LIN {X 0,Y 523.493,Z 544.016,A -85,B 0,C 180,E1 -4763.834,E2 -4763.834} C_VEL
LIN {X 0,Y 523.412,Z 548.835,A -85,B 0,C 180,E1 -4764.993,E2 -4764.993} C_VEL
LIN {X 0,Y 523.475,Z 552.534,A -85,B 0,C 180,E1 -4766.151,E2 -4766.151} C_VEL
LIN {X 0,Y 523.423,Z 554.433,A -85,B 0,C 180,E1 -4766.921,E2 -4766.921} C_VEL
LIN {X 0,Y 523.357,Z 555.854,A -85,B 0,C 180,E1 -4767.691,E2 -4767.691} C_VEL
LIN {X 0,Y 523.305,Z 557.491,A -85,B 0,C 180,E1 -4769.23,E2 -4769.23} C_VEL
LIN {X 0,Y 523.307,Z 557.714,A -85,B 0,C 180,E1 -4770,E2 -4770} C_VEL
LIN {X 0,Y 523.305,Z 557.495,A -85,B 0,C 180,E1 -4770.769,E2 -4770.769} C_VEL
LIN {X 0,Y 523.356,Z 555.866,A -85,B 0,C 180,E1 -4772.308,E2 -4772.308} C_VEL
LIN {X 0,Y 523.423,Z 554.448,A -85,B 0,C 180,E1 -4773.078,E2 -4773.078} C_VEL
LIN {X 0,Y 523.442,Z 551.453,A -85,B 0,C 180,E1 -4774.234,E2 -4774.234} C_VEL
LIN {X 0,Y 523.464,Z 547.399,A -85,B 0,C 180,E1 -4775.392,E2 -4775.392} C_VEL
LIN {X 0,Y 523.516,Z 542.074,A -85,B 0,C 180,E1 -4776.574,E2 -4776.574} C_VEL
LIN {X 0,Y 523.617,Z 535.63,A -85,B 0,C 180,E1 -4777.713,E2 -4777.713} C_VEL
LIN {X 0,Y 523.804,Z 527.471,A -85,B 0,C 180,E1 -4778.876,E2 -4778.876} C_VEL
LIN {X 0,Y 523.991,Z 519.167,A -85,B 0,C 180,E1 -4779.846,E2 -4779.846} C_VEL
LIN {X 0,Y 524.24,Z 509.058,A -85,B 0,C 180,E1 -4780.817,E2 -4780.817} C_VEL
LIN {X 0,Y 524.542,Z 497.688,A -85,B 0,C 180,E1 -4781.69,E2 -4781.69} C_VEL
LIN {X 0,Y 524.792,Z 486.52,A -85,B 0,C 180,E1 -4782.372,E2 -4782.372} C_VEL
LIN {X 0,Y 525.029,Z 475.334,A -85,B 0,C 180,E1 -4782.907,E2 -4782.907} C_VEL
LIN {X 0,Y 525.268,Z 462.202,A -85,B 0,C 180,E1 -4783.368,E2 -4783.368} C_VEL
LIN {X 0,Y 525.476,Z 449.138,A -85,B 0,C 180,E1 -4783.658,E2 -4783.658} C_VEL
LIN {X 0,Y 525.785,Z 353.498,A -85,B 0,C 180,E1 -4784.975,E2 -4784.975} C_VEL
LIN {X 0,Y 524.395,Z 341.8,A -85,B 0,C 180,E1 -4785.201,E2 -4785.201} C_VEL
LIN {X 0,Y 524.831,Z 315.783,A -85,B 0,C 180,E1 -4788.301,E2 -4788.301} C_VEL
LIN {X 0,Y 525.302,Z 288.649,A -85,B 0,C 180,E1 -4791.587,E2 -4791.587} C_VEL
LIN {X 0,Y 525.7,Z 266.745,A -85,B 0,C 180,E1 -4794.272,E2 -4794.272} C_VEL
LIN {X 0,Y 525.943,Z 250.474,A -85,B 0,C 180,E1 -4796.291,E2 -4796.291} C_VEL
LIN {X 0,Y 523.9,Z 240.345,A -85,B 0,C 180,E1 -4797.674,E2 -4797.674} C_VEL
LIN {X 0,Y 523.893,Z 240.226,A -85,B 0,C 180,E1 -4800.845,E2 -4800.845} C_VEL
LIN {X 0,Y 523.92,Z 240.225,A -85,B 0,C 180,E1 -4803.728,E2 -4803.728} C_VEL
LIN {X 0,Y 523.851,Z 240.227,A -85,B 0,C 180,E1 -4806.393,E2 -4806.393} C_VEL
LIN {X 0,Y 523.883,Z 240.228,A -85,B 0,C 180,E1 -4809.087,E2 -4809.087} C_VEL
LIN {X 0,Y 523.879,Z 240.223,A -85,B 0,C 180,E1 -4812.125,E2 -4812.125} C_VEL
LIN {X 0,Y 523.922,Z 240.226,A -85,B 0,C 180,E1 -4815.311,E2 -4815.311} C_VEL
LIN {X 0,Y 523.904,Z 240.222,A -85,B 0,C 180,E1 -4818.694,E2 -4818.694} C_VEL
LIN {X 0,Y 523.889,Z 240.222,A -85,B 0,C 180,E1 -4821.896,E2 -4821.896} C_VEL
LIN {X 0,Y 523.902,Z 240.227,A -85,B 0,C 180,E1 -4824.912,E2 -4824.912} C_VEL
LIN {X 0,Y 523.887,Z 240.223,A -85,B 0,C 180,E1 -4827.686,E2 -4827.686} C_VEL
LIN {X 0,Y 523.918,Z 240.223,A -85,B 0,C 180,E1 -4830.681,E2 -4830.681} C_VEL
LIN {X 0,Y 523.87,Z 240.225,A -85,B 0,C 180,E1 -4833.723,E2 -4833.723} C_VEL
LIN {X 0,Y 523.893,Z 240.223,A -85,B 0,C 180,E1 -4836.269,E2 -4836.269} C_VEL
LIN {X 0,Y 523.916,Z 240.226,A -85,B 0,C 180,E1 -4838.765,E2 -4838.765} C_VEL
LIN {X 0,Y 523.913,Z 240.222,A -85,B 0,C 180,E1 -4841.219,E2 -4841.219} C_VEL
LIN {X 0,Y 523.874,Z 240.224,A -85,B 0,C 180,E1 -4843.637,E2 -4843.637} C_VEL
LIN {X 0,Y 523.894,Z 240.222,A -85,B 0,C 180,E1 -4846.027,E2 -4846.027} C_VEL
LIN {X 0,Y 523.999,Z 240.213,A -85,B 0,C 180,E1 -4848.394,E2 -4848.394} C_VEL
LIN {X 0,Y 523.941,Z 240.215,A -85,B 0,C 180,E1 -4851.515,E2 -4851.515} C_VEL
LIN {X 0,Y 524.014,Z 240.216,A -85,B 0,C 180,E1 -4854.613,E2 -4854.613} C_VEL
LIN {X 0,Y 524.083,Z 240.198,A -85,B 0,C 180,E1 -4857.695,E2 -4857.695} C_VEL
LIN {X 0,Y 524.104,Z 240.2,A -85,B 0,C 180,E1 -4860.769,E2 -4860.769} C_VEL
LIN {X 0,Y 523.984,Z 240.211,A -85,B 0,C 180,E1 -4863.076,E2 -4863.076} C_VEL
LIN {X 0,Y 523.987,Z 240.215,A -85,B 0,C 180,E1 -4866.16,E2 -4866.16} C_VEL
LIN {X 0,Y 523.927,Z 240.217,A -85,B 0,C 180,E1 -4869.263,E2 -4869.263} C_VEL
LIN {X 0,Y 523.933,Z 240.224,A -85,B 0,C 180,E1 -4872.394,E2 -4872.394} C_VEL
LIN {X 0,Y 523.908,Z 240.22,A -85,B 0,C 180,E1 -4875.563,E2 -4875.563} C_VEL
LIN {X 0,Y 523.901,Z 240.226,A -85,B 0,C 180,E1 -4877.972,E2 -4877.972} C_VEL
LIN {X 0,Y 523.937,Z 240.221,A -85,B 0,C 180,E1 -4880.412,E2 -4880.412} C_VEL
LIN {X 0,Y 523.895,Z 240.222,A -85,B 0,C 180,E1 -4882.895,E2 -4882.895} C_VEL
LIN {X 0,Y 523.884,Z 240.224,A -85,B 0,C 180,E1 -4885.423,E2 -4885.423} C_VEL
LIN {X 0,Y 523.884,Z 240.231,A -85,B 0,C 180,E1 -4888.004,E2 -4888.004} C_VEL
LIN {X 0,Y 523.897,Z 240.221,A -85,B 0,C 180,E1 -4890.849,E2 -4890.849} C_VEL
LIN {X 0,Y 523.916,Z 240.224,A -85,B 0,C 180,E1 -4893.73,E2 -4893.73} C_VEL
LIN {X 0,Y 523.85,Z 240.229,A -85,B 0,C 180,E1 -4896.396,E2 -4896.396} C_VEL
LIN {X 0,Y 523.884,Z 240.223,A -85,B 0,C 180,E1 -4899.089,E2 -4899.089} C_VEL
LIN {X 0,Y 523.878,Z 240.228,A -85,B 0,C 180,E1 -4902.127,E2 -4902.127} C_VEL
LIN {X 0,Y 523.925,Z 240.22,A -85,B 0,C 180,E1 -4905.313,E2 -4905.313} C_VEL
LIN {X 0,Y 523.869,Z 240.225,A -85,B 0,C 180,E1 -4906.913,E2 -4906.913} C_VEL
LIN {X 0,Y 523.186,Z 240.316,A -85,B 0,C 180,E1 -4907.555,E2 -4907.555} C_VEL
LIN {X 0,Y 520.325,Z 240.672,A -85,B 0,C 180,E1 -4908.596,E2 -4908.596} C_VEL
LIN {X 0,Y 517.925,Z 240.97,A -85,B 0,C 180,E1 -4909.435,E2 -4909.435} C_VEL
LIN {X 0,Y 516.905,Z 241.096,A -85,B 0,C 180,E1 -4910.083,E2 -4910.083} C_VEL
LIN {X 0,Y 516.828,Z 241.103,A -85,B 0,C 180,E1 -4910.302,E2 -4910.302} C_VEL
LIN {X 0,Y 516.826,Z 241.103,A -85,B 0,C 180,E1 -4912.272,E2 -4912.272} C_VEL
LIN {X 0,Y 516.848,Z 241.102,A -85,B 0,C 180,E1 -4915.174,E2 -4915.174} C_VEL
LIN {X 0,Y 516.843,Z 241.103,A -85,B 0,C 180,E1 -4917.974,E2 -4917.974} C_VEL
LIN {X 0,Y 516.833,Z 241.101,A -85,B 0,C 180,E1 -4920.691,E2 -4920.691} C_VEL
LIN {X 0,Y 516.825,Z 241.109,A -85,B 0,C 180,E1 -4923.338,E2 -4923.338} C_VEL
LIN {X 0,Y 516.868,Z 241.099,A -85,B 0,C 180,E1 -4925.927,E2 -4925.927} C_VEL
LIN {X 0,Y 516.864,Z 241.097,A -85,B 0,C 180,E1 -4928.462,E2 -4928.462} C_VEL
LIN {X 0,Y 516.867,Z 241.1,A -85,B 0,C 180,E1 -4930.954,E2 -4930.954} C_VEL
LIN {X 0,Y 516.871,Z 241.104,A -85,B 0,C 180,E1 -4933.41,E2 -4933.41} C_VEL
LIN {X 0,Y 516.851,Z 241.1,A -85,B 0,C 180,E1 -4935.833,E2 -4935.833} C_VEL
LIN {X 0,Y 516.927,Z 241.09,A -85,B 0,C 180,E1 -4938.233,E2 -4938.233} C_VEL
LIN {X 0,Y 516.912,Z 241.1,A -85,B 0,C 180,E1 -4941.399,E2 -4941.399} C_VEL
LIN {X 0,Y 516.947,Z 241.206,A -85,B 0,C 180,E1 -4942.796,E2 -4942.796} C_VEL
LIN {X 0,Y 517.133,Z 242.04,A -85,B 0,C 180,E1 -4942.932,E2 -4942.932} C_VEL
LIN {X 0,Y 519.13,Z 247.934,A -85,B 0,C 180,E1 -4943.099,E2 -4943.099} C_VEL
LIN {X 0,Y 518.754,Z 330.215,A -85,B 0,C 180,E1 -4944.266,E2 -4944.266} C_VEL
LIN {X 0,Y 518.651,Z 343.83,A -85,B 0,C 180,E1 -4944.631,E2 -4944.631} C_VEL
LIN {X 0,Y 518.471,Z 356.587,A -85,B 0,C 180,E1 -4945.141,E2 -4945.141} C_VEL
LIN {X 0,Y 518.216,Z 368.942,A -85,B 0,C 180,E1 -4945.82,E2 -4945.82} C_VEL
LIN {X 0,Y 517.934,Z 379.943,A -85,B 0,C 180,E1 -4946.597,E2 -4946.597} C_VEL
LIN {X 0,Y 517.629,Z 389.885,A -85,B 0,C 180,E1 -4947.471,E2 -4947.471} C_VEL
LIN {X 0,Y 517.387,Z 398.828,A -85,B 0,C 180,E1 -4948.444,E2 -4948.444} C_VEL
LIN {X 0,Y 517.114,Z 407.548,A -85,B 0,C 180,E1 -4949.611,E2 -4949.611} C_VEL
LIN {X 0,Y 516.887,Z 414.584,A -85,B 0,C 180,E1 -4950.779,E2 -4950.779} C_VEL
LIN {X 0,Y 516.65,Z 420.23,A -85,B 0,C 180,E1 -4951.949,E2 -4951.949} C_VEL
LIN {X 0,Y 516.586,Z 424.66,A -85,B 0,C 180,E1 -4953.12,E2 -4953.12} C_VEL
LIN {X 0,Y 516.538,Z 427.004,A -85,B 0,C 180,E1 -4953.901,E2 -4953.901} C_VEL
LIN {X 0,Y 516.551,Z 428.921,A -85,B 0,C 180,E1 -4954.683,E2 -4954.683} C_VEL
LIN {X 0,Y 516.512,Z 430.446,A -85,B 0,C 180,E1 -4955.466,E2 -4955.466} C_VEL
LIN {X 0,Y 516.491,Z 431.912,A -85,B 0,C 180,E1 -4956.619,E2 -4956.619} C_VEL
LIN {X 0,Y 516.447,Z 432.547,A -85,B 0,C 180,E1 -4957.821,E2 -4957.821} C_VEL
LIN {X 0,Y 516.429,Z 432.486,A -85,B 0,C 180,E1 -4958.61,E2 -4958.61} C_VEL
LIN {X 0,Y 516.434,Z 432.004,A -85,B 0,C 180,E1 -4959.399,E2 -4959.399} C_VEL
LIN {X 0,Y 516.503,Z 429.826,A -85,B 0,C 180,E1 -4960.982,E2 -4960.982} C_VEL
LIN {X 0,Y 516.566,Z 427.084,A -85,B 0,C 180,E1 -4962.174,E2 -4962.174} C_VEL
LIN {X 0,Y 516.626,Z 423.297,A -85,B 0,C 180,E1 -4963.371,E2 -4963.371} C_VEL
LIN {X 0,Y 516.789,Z 418.342,A -85,B 0,C 180,E1 -4964.571,E2 -4964.571} C_VEL
LIN {X 0,Y 516.966,Z 412.054,A -85,B 0,C 180,E1 -4965.777,E2 -4965.777} C_VEL
LIN {X 0,Y 517.236,Z 404.087,A -85,B 0,C 180,E1 -4966.986,E2 -4966.986} C_VEL
LIN {X 0,Y 517.498,Z 395.21,A -85,B 0,C 180,E1 -4968.074,E2 -4968.074} C_VEL
LIN {X 0,Y 517.757,Z 385.794,A -85,B 0,C 180,E1 -4969.012,E2 -4969.012} C_VEL
LIN {X 0,Y 518.036,Z 375.687,A -85,B 0,C 180,E1 -4969.826,E2 -4969.826} C_VEL
LIN {X 0,Y 518.351,Z 364.124,A -85,B 0,C 180,E1 -4970.563,E2 -4970.563} C_VEL
LIN {X 0,Y 518.559,Z 352.167,A -85,B 0,C 180,E1 -4971.152,E2 -4971.152} C_VEL
LIN {X 0,Y 518.727,Z 339.918,A -85,B 0,C 180,E1 -4971.588,E2 -4971.588} C_VEL
LIN {X 0,Y 518.821,Z 326.93,A -85,B 0,C 180,E1 -4971.884,E2 -4971.884} C_VEL
LIN {X 0,Y 519.144,Z 248.098,A -85,B 0,C 180,E1 -4972.991,E2 -4972.991} C_VEL
LIN {X 0,Y 517.024,Z 241.898,A -85,B 0,C 180,E1 -4973.175,E2 -4973.175} C_VEL
LIN {X 0,Y 516.887,Z 241.164,A -85,B 0,C 180,E1 -4973.329,E2 -4973.329} C_VEL
LIN {X 0,Y 516.882,Z 241.1,A -85,B 0,C 180,E1 -4976.181,E2 -4976.181} C_VEL
LIN {X 0,Y 516.909,Z 241.093,A -85,B 0,C 180,E1 -4979.522,E2 -4979.522} C_VEL
LIN {X 0,Y 516.896,Z 241.094,A -85,B 0,C 180,E1 -4982.542,E2 -4982.542} C_VEL
LIN {X 0,Y 516.86,Z 241.091,A -85,B 0,C 180,E1 -4985.328,E2 -4985.328} C_VEL
LIN {X 0,Y 516.873,Z 241.101,A -85,B 0,C 180,E1 -4988.716,E2 -4988.716} C_VEL
LIN {X 0,Y 516.881,Z 241.093,A -85,B 0,C 180,E1 -4991.778,E2 -4991.778} C_VEL
LIN {X 0,Y 516.894,Z 241.096,A -85,B 0,C 180,E1 -4995.006,E2 -4995.006} C_VEL
LIN {X 0,Y 516.852,Z 241.104,A -85,B 0,C 180,E1 -4998.405,E2 -4998.405} C_VEL
LIN {X 0,Y 516.87,Z 241.094,A -85,B 0,C 180,E1 -5001.283,E2 -5001.283} C_VEL
LIN {X 0,Y 516.849,Z 241.104,A -85,B 0,C 180,E1 -5004.672,E2 -5004.672} C_VEL
LIN {X 0,Y 516.89,Z 241.094,A -85,B 0,C 180,E1 -5007.456,E2 -5007.456} C_VEL
LIN {X 0,Y 516.915,Z 241.09,A -85,B 0,C 180,E1 -5010.695,E2 -5010.695} C_VEL
LIN {X 0,Y 516.882,Z 241.1,A -85,B 0,C 180,E1 -5013.816,E2 -5013.816} C_VEL
LIN {X 0,Y 516.852,Z 241.091,A -85,B 0,C 180,E1 -5016.775,E2 -5016.775} C_VEL
LIN {X 0,Y 516.931,Z 241.083,A -85,B 0,C 180,E1 -5019.732,E2 -5019.732} C_VEL
LIN {X 0,Y 516.886,Z 241.096,A -85,B 0,C 180,E1 -5022.594,E2 -5022.594} C_VEL
LIN {X 0,Y 516.928,Z 241.087,A -85,B 0,C 180,E1 -5025.029,E2 -5025.029} C_VEL
LIN {X 0,Y 516.959,Z 241.089,A -85,B 0,C 180,E1 -5028.233,E2 -5028.233} C_VEL
LIN {X 0,Y 516.921,Z 241.089,A -85,B 0,C 180,E1 -5031.399,E2 -5031.399} C_VEL
LIN {X 0,Y 516.977,Z 241.083,A -85,B 0,C 180,E1 -5034.539,E2 -5034.539} C_VEL
LIN {X 0,Y 517.062,Z 241.078,A -85,B 0,C 180,E1 -5037.663,E2 -5037.663} C_VEL
LIN {X 0,Y 517.053,Z 241.077,A -85,B 0,C 180,E1 -5040,E2 -5040} C_VEL
LIN {X 0,Y 517.063,Z 241.071,A -85,B 0,C 180,E1 -5042.337,E2 -5042.337} C_VEL
LIN {X 0,Y 516.972,Z 241.092,A -85,B 0,C 180,E1 -5045.46,E2 -5045.46} C_VEL
LIN {X 0,Y 516.941,Z 241.086,A -85,B 0,C 180,E1 -5048.601,E2 -5048.601} C_VEL
LIN {X 0,Y 516.944,Z 241.088,A -85,B 0,C 180,E1 -5051.807,E2 -5051.807} C_VEL
LIN {X 0,Y 516.927,Z 241.094,A -85,B 0,C 180,E1 -5055.142,E2 -5055.142} C_VEL
LIN {X 0,Y 516.901,Z 241.091,A -85,B 0,C 180,E1 -5058.223,E2 -5058.223} C_VEL
LIN {X 0,Y 516.893,Z 241.096,A -85,B 0,C 180,E1 -5060.702,E2 -5060.702} C_VEL
LIN {X 0,Y 516.847,Z 241.107,A -85,B 0,C 180,E1 -5063.225,E2 -5063.225} C_VEL
LIN {X 0,Y 516.871,Z 241.094,A -85,B 0,C 180,E1 -5066.182,E2 -5066.182} C_VEL
LIN {X 0,Y 516.891,Z 241.1,A -85,B 0,C 180,E1 -5069.306,E2 -5069.306} C_VEL
LIN {X 0,Y 516.885,Z 241.097,A -85,B 0,C 180,E1 -5072.543,E2 -5072.543} C_VEL
LIN {X 0,Y 516.845,Z 241.104,A -85,B 0,C 180,E1 -5075.328,E2 -5075.328} C_VEL
LIN {X 0,Y 516.866,Z 241.101,A -85,B 0,C 180,E1 -5078.717,E2 -5078.717} C_VEL
LIN {X 0,Y 516.839,Z 241.101,A -85,B 0,C 180,E1 -5081.783,E2 -5081.783} C_VEL
LIN {X 0,Y 516.892,Z 241.1,A -85,B 0,C 180,E1 -5085.007,E2 -5085.007} C_VEL
LIN {X 0,Y 516.843,Z 241.105,A -85,B 0,C 180,E1 -5088.408,E2 -5088.408} C_VEL
LIN {X 0,Y 516.849,Z 241.099,A -85,B 0,C 180,E1 -5091.282,E2 -5091.282} C_VEL
LIN {X 0,Y 516.846,Z 241.101,A -85,B 0,C 180,E1 -5094.674,E2 -5094.674} C_VEL
LIN {X 0,Y 516.865,Z 241.097,A -85,B 0,C 180,E1 -5097.462,E2 -5097.462} C_VEL
LIN {X 0,Y 516.836,Z 241.104,A -85,B 0,C 180,E1 -5100.491,E2 -5100.491} C_VEL
LIN {X 0,Y 516.888,Z 241.337,A -85,B 0,C 180,E1 -5102.193,E2 -5102.193} C_VEL
LIN {X 0,Y 518.985,Z 252.032,A -85,B 0,C 180,E1 -5103.673,E2 -5103.673} C_VEL
LIN {X 0,Y 518.594,Z 273.99,A -85,B 0,C 180,E1 -5106.436,E2 -5106.436} C_VEL
LIN {X 0,Y 518.064,Z 300.994,A -85,B 0,C 180,E1 -5109.768,E2 -5109.768} C_VEL
LIN {X 0,Y 517.58,Z 326.077,A -85,B 0,C 180,E1 -5112.822,E2 -5112.822} C_VEL
LIN {X 0,Y 517.417,Z 341.054,A -85,B 0,C 180,E1 -5114.604,E2 -5114.604} C_VEL
LIN {X 0,Y 519.004,Z 355.896,A -85,B 0,C 180,E1 -5114.871,E2 -5114.871} C_VEL
LIN {X 0,Y 518.551,Z 451,A -85,B 0,C 180,E1 -5116.205,E2 -5116.205} C_VEL
LIN {X 0,Y 518.275,Z 464.373,A -85,B 0,C 180,E1 -5116.547,E2 -5116.547} C_VEL
LIN {X 0,Y 518.048,Z 476.648,A -85,B 0,C 180,E1 -5117.015,E2 -5117.015} C_VEL
LIN {X 0,Y 517.724,Z 488.312,A -85,B 0,C 180,E1 -5117.61,E2 -5117.61} C_VEL
LIN {X 0,Y 517.458,Z 499.483,A -85,B 0,C 180,E1 -5118.344,E2 -5118.344} C_VEL
LIN {X 0,Y 517.155,Z 510.292,A -85,B 0,C 180,E1 -5119.23,E2 -5119.23} C_VEL
LIN {X 0,Y 516.884,Z 520.05,A -85,B 0,C 180,E1 -5120.214,E2 -5120.214} C_VEL
LIN {X 0,Y 516.695,Z 528.067,A -85,B 0,C 180,E1 -5121.198,E2 -5121.198} C_VEL
LIN {X 0,Y 516.54,Z 535.913,A -85,B 0,C 180,E1 -5122.377,E2 -5122.377} C_VEL
LIN {X 0,Y 516.404,Z 541.789,A -85,B 0,C 180,E1 -5123.462,E2 -5123.462} C_VEL
LIN {X 0,Y 516.405,Z 546.518,A -85,B 0,C 180,E1 -5124.533,E2 -5124.533} C_VEL
LIN {X 0,Y 516.369,Z 550.577,A -85,B 0,C 180,E1 -5125.707,E2 -5125.707} C_VEL
LIN {X 0,Y 516.364,Z 553.578,A -85,B 0,C 180,E1 -5126.879,E2 -5126.879} C_VEL
LIN {X 0,Y 516.302,Z 555.002,A -85,B 0,C 180,E1 -5127.659,E2 -5127.659} C_VEL
LIN {X 0,Y 516.254,Z 556.642,A -85,B 0,C 180,E1 -5129.22,E2 -5129.22} C_VEL
LIN {X 0,Y 516.259,Z 556.866,A -85,B 0,C 180,E1 -5130,E2 -5130} C_VEL
LIN {X 0,Y 516.254,Z 556.647,A -85,B 0,C 180,E1 -5130.78,E2 -5130.78} C_VEL
LIN {X 0,Y 516.301,Z 555.019,A -85,B 0,C 180,E1 -5132.34,E2 -5132.34} C_VEL
LIN {X 0,Y 516.364,Z 553.601,A -85,B 0,C 180,E1 -5133.12,E2 -5133.12} C_VEL
LIN {X 0,Y 516.368,Z 550.604,A -85,B 0,C 180,E1 -5134.293,E2 -5134.293} C_VEL
LIN {X 0,Y 516.404,Z 546.55,A -85,B 0,C 180,E1 -5135.466,E2 -5135.466} C_VEL
LIN {X 0,Y 516.485,Z 540.477,A -85,B 0,C 180,E1 -5136.808,E2 -5136.808} C_VEL
LIN {X 0,Y 516.583,Z 533.521,A -85,B 0,C 180,E1 -5138.015,E2 -5138.015} C_VEL
LIN {X 0,Y 516.751,Z 525.1,A -85,B 0,C 180,E1 -5139.195,E2 -5139.195} C_VEL
LIN {X 0,Y 516.975,Z 516.483,A -85,B 0,C 180,E1 -5140.179,E2 -5140.179} C_VEL
LIN {X 0,Y 517.247,Z 505.853,A -85,B 0,C 180,E1 -5141.163,E2 -5141.163} C_VEL
LIN {X 0,Y 517.562,Z 495.038,A -85,B 0,C 180,E1 -5141.973,E2 -5141.973} C_VEL
LIN {X 0,Y 517.853,Z 483.879,A -85,B 0,C 180,E1 -5142.64,E2 -5142.64} C_VEL
LIN {X 0,Y 518.121,Z 472.11,A -85,B 0,C 180,E1 -5143.182,E2 -5143.182} C_VEL
LIN {X 0,Y 518.394,Z 458.587,A -85,B 0,C 180,E1 -5143.624,E2 -5143.624} C_VEL
LIN {X 0,Y 518.632,Z 445.241,A -85,B 0,C 180,E1 -5143.892,E2 -5143.892} C_VEL
LIN {X 0,Y 518.848,Z 353.499,A -85,B 0,C 180,E1 -5145.168,E2 -5145.168} C_VEL
LIN {X 0,Y 517.4,Z 341.07,A -85,B 0,C 180,E1 -5145.402,E2 -5145.402} C_VEL
LIN {X 0,Y 517.854,Z 314.597,A -85,B 0,C 180,E1 -5148.597,E2 -5148.597} C_VEL
LIN {X 0,Y 518.306,Z 289.478,A -85,B 0,C 180,E1 -5151.684,E2 -5151.684} C_VEL
LIN {X 0,Y 518.715,Z 269.237,A -85,B 0,C 180,E1 -5154.195,E2 -5154.195} C_VEL
LIN {X 0,Y 519.031,Z 252.234,A -85,B 0,C 180,E1 -5156.324,E2 -5156.324} C_VEL
LIN {X 0,Y 516.85,Z 241.238,A -85,B 0,C 180,E1 -5157.838,E2 -5157.838} C_VEL
LIN {X 0,Y 516.844,Z 241.104,A -85,B 0,C 180,E1 -5161.055,E2 -5161.055} C_VEL
LIN {X 0,Y 516.875,Z 241.1,A -85,B 0,C 180,E1 -5163.96,E2 -5163.96} C_VEL
LIN {X 0,Y 516.799,Z 241.106,A -85,B 0,C 180,E1 -5166.751,E2 -5166.751} C_VEL
LIN {X 0,Y 516.827,Z 241.105,A -85,B 0,C 180,E1 -5169.725,E2 -5169.725} C_VEL
LIN {X 0,Y 516.829,Z 241.104,A -85,B 0,C 180,E1 -5172.835,E2 -5172.835} C_VEL
LIN {X 0,Y 516.888,Z 241.099,A -85,B 0,C 180,E1 -5175.006,E2 -5175.006} C_VEL
LIN {X 0,Y 516.84,Z 241.1,A -85,B 0,C 180,E1 -5178.406,E2 -5178.406} C_VEL
LIN {X 0,Y 516.86,Z 241.104,A -85,B 0,C 180,E1 -5181.282,E2 -5181.282} C_VEL
LIN {X 0,Y 516.84,Z 241.103,A -85,B 0,C 180,E1 -5184.672,E2 -5184.672} C_VEL
LIN {X 0,Y 516.852,Z 241.102,A -85,B 0,C 180,E1 -5187.462,E2 -5187.462} C_VEL
LIN {X 0,Y 516.885,Z 241.099,A -85,B 0,C 180,E1 -5190.693,E2 -5190.693} C_VEL
LIN {X 0,Y 516.847,Z 241.099,A -85,B 0,C 180,E1 -5193.822,E2 -5193.822} C_VEL
LIN {X 0,Y 516.842,Z 241.107,A -85,B 0,C 180,E1 -5196.775,E2 -5196.775} C_VEL
LIN {X 0,Y 516.893,Z 241.093,A -85,B 0,C 180,E1 -5199.741,E2 -5199.741} C_VEL
LIN {X 0,Y 516.87,Z 241.102,A -85,B 0,C 180,E1 -5202.594,E2 -5202.594} C_VEL
LIN {X 0,Y 516.916,Z 241.095,A -85,B 0,C 180,E1 -5205.029,E2 -5205.029} C_VEL
LIN {X 0,Y 516.953,Z 241.089,A -85,B 0,C 180,E1 -5208.233,E2 -5208.233} C_VEL
LIN {X 0,Y 516.912,Z 241.092,A -85,B 0,C 180,E1 -5211.399,E2 -5211.399} C_VEL
LIN {X 0,Y 516.964,Z 241.093,A -85,B 0,C 180,E1 -5214.539,E2 -5214.539} C_VEL
LIN {X 0,Y 517.055,Z 241.073,A -85,B 0,C 180,E1 -5217.663,E2 -5217.663} C_VEL
LIN {X 0,Y 517.074,Z 241.076,A -85,B 0,C 180,E1 -5220.779,E2 -5220.779} C_VEL
LIN {X 0,Y 516.927,Z 241.09,A -85,B 0,C 180,E1 -5223.118,E2 -5223.118} C_VEL
LIN {X 0,Y 516.954,Z 241.092,A -85,B 0,C 180,E1 -5226.244,E2 -5226.244} C_VEL
LIN {X 0,Y 516.889,Z 241.094,A -85,B 0,C 180,E1 -5229.391,E2 -5229.391} C_VEL
LIN {X 0,Y 516.886,Z 241.099,A -85,B 0,C 180,E1 -5232.565,E2 -5232.565} C_VEL
LIN {X 0,Y 516.93,Z 241.089,A -85,B 0,C 180,E1 -5235.146,E2 -5235.146} C_VEL
LIN {X 0,Y 516.862,Z 241.106,A -85,B 0,C 180,E1 -5238.225,E2 -5238.225} C_VEL
LIN {X 0,Y 516.887,Z 241.096,A -85,B 0,C 180,E1 -5240.703,E2 -5240.703} C_VEL
LIN {X 0,Y 516.845,Z 241.099,A -85,B 0,C 180,E1 -5243.225,E2 -5243.225} C_VEL
LIN {X 0,Y 516.856,Z 241.106,A -85,B 0,C 180,E1 -5246.18,E2 -5246.18} C_VEL
LIN {X 0,Y 516.892,Z 241.094,A -85,B 0,C 180,E1 -5249.307,E2 -5249.307} C_VEL
LIN {X 0,Y 516.839,Z 241.109,A -85,B 0,C 180,E1 -5252.028,E2 -5252.028} C_VEL
LIN {X 0,Y 516.86,Z 241.098,A -85,B 0,C 180,E1 -5254.827,E2 -5254.827} C_VEL
LIN {X 0,Y 516.842,Z 241.108,A -85,B 0,C 180,E1 -5257.94,E2 -5257.94} C_VEL
LIN {X 0,Y 516.811,Z 241.104,A -85,B 0,C 180,E1 -5260.749,E2 -5260.749} C_VEL
LIN {X 0,Y 516.853,Z 241.106,A -85,B 0,C 180,E1 -5263.907,E2 -5263.907} C_VEL
LIN {X 0,Y 516.854,Z 241.102,A -85,B 0,C 180,E1 -5266.111,E2 -5266.111} C_VEL
LIN {X 0,Y 516.816,Z 241.106,A -85,B 0,C 180,E1 -5269.253,E2 -5269.253} C_VEL
LIN {X 0,Y 516.828,Z 241.103,A -85,B 0,C 180,E1 -5270.302,E2 -5270.302} C_VEL
LIN {X 0,Y 516.174,Z 241.184,A -85,B 0,C 180,E1 -5270.952,E2 -5270.952} C_VEL
LIN {X 0,Y 513.317,Z 241.548,A -85,B 0,C 180,E1 -5272.008,E2 -5272.008} C_VEL
LIN {X 0,Y 510.89,Z 241.855,A -85,B 0,C 180,E1 -5272.858,E2 -5272.858} C_VEL
LIN {X 0,Y 509.843,Z 241.982,A -85,B 0,C 180,E1 -5273.515,E2 -5273.515} C_VEL
LIN {X 0,Y 509.756,Z 241.99,A -85,B 0,C 180,E1 -5273.738,E2 -5273.738} C_VEL
LIN {X 0,Y 509.821,Z 241.974,A -85,B 0,C 180,E1 -5276.538,E2 -5276.538} C_VEL
LIN {X 0,Y 509.8,Z 241.983,A -85,B 0,C 180,E1 -5279.332,E2 -5279.332} C_VEL
LIN {X 0,Y 509.822,Z 241.976,A -85,B 0,C 180,E1 -5282.051,E2 -5282.051} C_VEL
LIN {X 0,Y 509.781,Z 241.98,A -85,B 0,C 180,E1 -5284.7,E2 -5284.7} C_VEL
LIN {X 0,Y 509.825,Z 241.982,A -85,B 0,C 180,E1 -5287.46,E2 -5287.46} C_VEL
LIN {X 0,Y 509.845,Z 241.974,A -85,B 0,C 180,E1 -5289.843,E2 -5289.843} C_VEL
LIN {X 0,Y 509.845,Z 241.978,A -85,B 0,C 180,E1 -5293.174,E2 -5293.174} C_VEL
LIN {X 0,Y 509.817,Z 241.979,A -85,B 0,C 180,E1 -5295.633,E2 -5295.633} C_VEL
LIN {X 0,Y 509.892,Z 241.967,A -85,B 0,C 180,E1 -5298.132,E2 -5298.132} C_VEL
LIN {X 0,Y 509.864,Z 241.977,A -85,B 0,C 180,E1 -5301.279,E2 -5301.279} C_VEL
LIN {X 0,Y 509.938,Z 242.129,A -85,B 0,C 180,E1 -5302.601,E2 -5302.601} C_VEL
LIN {X 0,Y 510.121,Z 243.044,A -85,B 0,C 180,E1 -5302.73,E2 -5302.73} C_VEL
LIN {X 0,Y 512.347,Z 249.633,A -85,B 0,C 180,E1 -5302.909,E2 -5302.909} C_VEL
LIN {X 0,Y 511.907,Z 330.464,A -85,B 0,C 180,E1 -5304.066,E2 -5304.066} C_VEL
LIN {X 0,Y 511.792,Z 343.54,A -85,B 0,C 180,E1 -5304.41,E2 -5304.41} C_VEL
LIN {X 0,Y 511.618,Z 356.611,A -85,B 0,C 180,E1 -5304.927,E2 -5304.927} C_VEL
LIN {X 0,Y 511.373,Z 368.416,A -85,B 0,C 180,E1 -5305.567,E2 -5305.567} C_VEL
LIN {X 0,Y 511.05,Z 379.673,A -85,B 0,C 180,E1 -5306.354,E2 -5306.354} C_VEL
LIN {X 0,Y 510.718,Z 389.823,A -85,B 0,C 180,E1 -5307.24,E2 -5307.24} C_VEL
LIN {X 0,Y 510.462,Z 398.967,A -85,B 0,C 180,E1 -5308.225,E2 -5308.225} C_VEL
LIN {X 0,Y 510.156,Z 407.807,A -85,B 0,C 180,E1 -5309.408,E2 -5309.408} C_VEL
LIN {X 0,Y 509.901,Z 414.947,A -85,B 0,C 180,E1 -5310.593,E2 -5310.593} C_VEL
LIN {X 0,Y 509.63,Z 421.518,A -85,B 0,C 180,E1 -5311.976,E2 -5311.976} C_VEL
LIN {X 0,Y 509.553,Z 425.847,A -85,B 0,C 180,E1 -5313.163,E2 -5313.163} C_VEL
LIN {X 0,Y 509.502,Z 428.14,A -85,B 0,C 180,E1 -5313.955,E2 -5313.955} C_VEL
LIN {X 0,Y 509.53,Z 430.007,A -85,B 0,C 180,E1 -5314.747,E2 -5314.747} C_VEL
LIN {X 0,Y 509.487,Z 431.471,A -85,B 0,C 180,E1 -5315.541,E2 -5315.541} C_VEL
LIN {X 0,Y 509.455,Z 433.141,A -85,B 0,C 180,E1 -5317.132,E2 -5317.132} C_VEL
LIN {X 0,Y 509.406,Z 433.418,A -85,B 0,C 180,E1 -5317.93,E2 -5317.93} C_VEL
LIN {X 0,Y 509.403,Z 433.292,A -85,B 0,C 180,E1 -5318.729,E2 -5318.729} C_VEL
LIN {X 0,Y 509.382,Z 431.811,A -85,B 0,C 180,E1 -5320.333,E2 -5320.333} C_VEL
LIN {X 0,Y 509.539,Z 429.313,A -85,B 0,C 180,E1 -5321.678,E2 -5321.678} C_VEL
LIN {X 0,Y 509.602,Z 425.167,A -85,B 0,C 180,E1 -5323.153,E2 -5323.153} C_VEL
LIN {X 0,Y 509.719,Z 420.497,A -85,B 0,C 180,E1 -5324.37,E2 -5324.37} C_VEL
LIN {X 0,Y 509.961,Z 413.519,A -85,B 0,C 180,E1 -5325.774,E2 -5325.774} C_VEL
LIN {X 0,Y 510.192,Z 407.026,A -85,B 0,C 180,E1 -5326.815,E2 -5326.815} C_VEL
LIN {X 0,Y 510.455,Z 398.782,A -85,B 0,C 180,E1 -5327.902,E2 -5327.902} C_VEL
LIN {X 0,Y 510.795,Z 388.693,A -85,B 0,C 180,E1 -5328.969,E2 -5328.969} C_VEL
LIN {X 0,Y 511.1,Z 377.77,A -85,B 0,C 180,E1 -5329.897,E2 -5329.897} C_VEL
LIN {X 0,Y 511.465,Z 366.226,A -85,B 0,C 180,E1 -5330.662,E2 -5330.662} C_VEL
LIN {X 0,Y 511.684,Z 353.887,A -85,B 0,C 180,E1 -5331.292,E2 -5331.292} C_VEL
LIN {X 0,Y 511.852,Z 341.221,A -85,B 0,C 180,E1 -5331.76,E2 -5331.76} C_VEL
LIN {X 0,Y 511.99,Z 327.788,A -85,B 0,C 180,E1 -5332.072,E2 -5332.072} C_VEL
LIN {X 0,Y 512.276,Z 249.335,A -85,B 0,C 180,E1 -5333.192,E2 -5333.192} C_VEL
LIN {X 0,Y 509.979,Z 242.763,A -85,B 0,C 180,E1 -5333.394,E2 -5333.394} C_VEL
LIN {X 0,Y 509.866,Z 242.03,A -85,B 0,C 180,E1 -5333.561,E2 -5333.561} C_VEL
LIN {X 0,Y 509.825,Z 241.983,A -85,B 0,C 180,E1 -5337.059,E2 -5337.059} C_VEL
LIN {X 0,Y 509.859,Z 241.971,A -85,B 0,C 180,E1 -5339.751,E2 -5339.751} C_VEL
LIN {X 0,Y 509.847,Z 241.976,A -85,B 0,C 180,E1 -5342.768,E2 -5342.768} C_VEL
LIN {X 0,Y 509.82,Z 241.967,A -85,B 0,C 180,E1 -5345.577,E2 -5345.577} C_VEL
LIN {X 0,Y 509.816,Z 241.973,A -85,B 0,C 180,E1 -5348.34,E2 -5348.34} C_VEL
LIN {X 0,Y 509.829,Z 241.972,A -85,B 0,C 180,E1 -5351.427,E2 -5351.427} C_VEL
LIN {X 0,Y 509.838,Z 241.979,A -85,B 0,C 180,E1 -5354.669,E2 -5354.669} C_VEL
LIN {X 0,Y 509.788,Z 241.975,A -85,B 0,C 180,E1 -5357.505,E2 -5357.505} C_VEL
LIN {X 0,Y 509.829,Z 241.976,A -85,B 0,C 180,E1 -5360.645,E2 -5360.645} C_VEL
LIN {X 0,Y 509.776,Z 241.976,A -85,B 0,C 180,E1 -5363.642,E2 -5363.642} C_VEL
LIN {X 0,Y 509.848,Z 241.976,A -85,B 0,C 180,E1 -5366.538,E2 -5366.538} C_VEL
LIN {X 0,Y 509.838,Z 241.963,A -85,B 0,C 180,E1 -5369.333,E2 -5369.333} C_VEL
LIN {X 0,Y 509.829,Z 241.976,A -85,B 0,C 180,E1 -5372.05,E2 -5372.05} C_VEL
LIN {X 0,Y 509.808,Z 241.977,A -85,B 0,C 180,E1 -5374.7,E2 -5374.7} C_VEL
LIN {X 0,Y 509.819,Z 241.967,A -85,B 0,C 180,E1 -5377.458,E2 -5377.458} C_VEL
LIN {X 0,Y 509.908,Z 241.959,A -85,B 0,C 180,E1 -5379.844,E2 -5379.844} C_VEL
LIN {X 0,Y 509.853,Z 241.971,A -85,B 0,C 180,E1 -5383.173,E2 -5383.173} C_VEL
LIN {X 0,Y 509.845,Z 241.973,A -85,B 0,C 180,E1 -5385.633,E2 -5385.633} C_VEL
LIN {X 0,Y 509.902,Z 241.964,A -85,B 0,C 180,E1 -5388.874,E2 -5388.874} C_VEL
LIN {X 0,Y 509.868,Z 241.974,A -85,B 0,C 180,E1 -5392.077,E2 -5392.077} C_VEL
LIN {X 0,Y 509.932,Z 241.961,A -85,B 0,C 180,E1 -5394.464,E2 -5394.464} C_VEL
LIN {X 0,Y 510.031,Z 241.953,A -85,B 0,C 180,E1 -5397.631,E2 -5397.631} C_VEL
LIN {X 0,Y 510.022,Z 241.952,A -85,B 0,C 180,E1 -5400,E2 -5400} C_VEL
LIN {X 0,Y 510.034,Z 241.946,A -85,B 0,C 180,E1 -5402.369,E2 -5402.369} C_VEL
LIN {X 0,Y 509.924,Z 241.969,A -85,B 0,C 180,E1 -5405.536,E2 -5405.536} C_VEL
LIN {X 0,Y 509.889,Z 241.964,A -85,B 0,C 180,E1 -5408.721,E2 -5408.721} C_VEL
LIN {X 0,Y 509.896,Z 241.965,A -85,B 0,C 180,E1 -5411.932,E2 -5411.932} C_VEL
LIN {X 0,Y 509.887,Z 241.972,A -85,B 0,C 180,E1 -5415.242,E2 -5415.242} C_VEL
LIN {X 0,Y 509.845,Z 241.97,A -85,B 0,C 180,E1 -5418.484,E2 -5418.484} C_VEL
LIN {X 0,Y 509.835,Z 241.979,A -85,B 0,C 180,E1 -5421.002,E2 -5421.002} C_VEL
LIN {X 0,Y 509.809,Z 241.981,A -85,B 0,C 180,E1 -5423.564,E2 -5423.564} C_VEL
LIN {X 0,Y 509.807,Z 241.974,A -85,B 0,C 180,E1 -5426.356,E2 -5426.356} C_VEL
LIN {X 0,Y 509.824,Z 241.973,A -85,B 0,C 180,E1 -5428.848,E2 -5428.848} C_VEL
LIN {X 0,Y 509.79,Z 241.98,A -85,B 0,C 180,E1 -5431.592,E2 -5431.592} C_VEL
LIN {X 0,Y 509.832,Z 241.968,A -85,B 0,C 180,E1 -5434.2,E2 -5434.2} C_VEL
LIN {X 0,Y 509.776,Z 241.982,A -85,B 0,C 180,E1 -5437.344,E2 -5437.344} C_VEL
LIN {X 0,Y 509.808,Z 241.978,A -85,B 0,C 180,E1 -5440.385,E2 -5440.385} C_VEL
LIN {X 0,Y 509.787,Z 241.979,A -85,B 0,C 180,E1 -5443.575,E2 -5443.575} C_VEL
LIN {X 0,Y 509.787,Z 241.983,A -85,B 0,C 180,E1 -5446.425,E2 -5446.425} C_VEL
LIN {X 0,Y 509.788,Z 241.976,A -85,B 0,C 180,E1 -5449.614,E2 -5449.614} C_VEL
LIN {X 0,Y 509.76,Z 241.99,A -85,B 0,C 180,E1 -5452.655,E2 -5452.655} C_VEL
LIN {X 0,Y 509.836,Z 241.973,A -85,B 0,C 180,E1 -5455.801,E2 -5455.801} C_VEL
LIN {X 0,Y 509.813,Z 241.981,A -85,B 0,C 180,E1 -5458.727,E2 -5458.727} C_VEL
LIN {X 0,Y 509.803,Z 242.161,A -85,B 0,C 180,E1 -5461.977,E2 -5461.977} C_VEL
LIN {X 0,Y 512.065,Z 253.338,A -85,B 0,C 180,E1 -5463.561,E2 -5463.561} C_VEL
LIN {X 0,Y 511.648,Z 274.864,A -85,B 0,C 180,E1 -5466.311,E2 -5466.311} C_VEL
LIN {X 0,Y 511.061,Z 300.683,A -85,B 0,C 180,E1 -5469.548,E2 -5469.548} C_VEL
LIN {X 0,Y 510.538,Z 326.859,A -85,B 0,C 180,E1 -5472.785,E2 -5472.785} C_VEL
LIN {X 0,Y 510.345,Z 340.076,A -85,B 0,C 180,E1 -5474.382,E2 -5474.382} C_VEL
LIN {X 0,Y 512.127,Z 356.552,A -85,B 0,C 180,E1 -5474.685,E2 -5474.685} C_VEL
LIN {X 0,Y 511.655,Z 450.112,A -85,B 0,C 180,E1 -5476.015,E2 -5476.015} C_VEL
LIN {X 0,Y 511.322,Z 463.485,A -85,B 0,C 180,E1 -5476.361,E2 -5476.361} C_VEL
LIN {X 0,Y 511.053,Z 476.898,A -85,B 0,C 180,E1 -5476.885,E2 -5476.885} C_VEL
LIN {X 0,Y 510.668,Z 489.28,A -85,B 0,C 180,E1 -5477.551,E2 -5477.551} C_VEL
LIN {X 0,Y 510.355,Z 501.22,A -85,B 0,C 180,E1 -5478.381,E2 -5478.381} C_VEL
LIN {X 0,Y 510.054,Z 511.565,A -85,B 0,C 180,E1 -5479.28,E2 -5479.28} C_VEL
LIN {X 0,Y 509.765,Z 520.884,A -85,B 0,C 180,E1 -5480.277,E2 -5480.277} C_VEL
LIN {X 0,Y 509.562,Z 529.986,A -85,B 0,C 180,E1 -5481.473,E2 -5481.473} C_VEL
LIN {X 0,Y 509.43,Z 537.327,A -85,B 0,C 180,E1 -5482.668,E2 -5482.668} C_VEL
LIN {X 0,Y 509.314,Z 542.284,A -85,B 0,C 180,E1 -5483.662,E2 -5483.662} C_VEL
LIN {X 0,Y 509.278,Z 547.115,A -85,B 0,C 180,E1 -5484.853,E2 -5484.853} C_VEL
LIN {X 0,Y 509.336,Z 550.819,A -85,B 0,C 180,E1 -5486.044,E2 -5486.044} C_VEL
LIN {X 0,Y 509.307,Z 552.724,A -85,B 0,C 180,E1 -5486.836,E2 -5486.836} C_VEL
LIN {X 0,Y 509.247,Z 554.149,A -85,B 0,C 180,E1 -5487.627,E2 -5487.627} C_VEL
LIN {X 0,Y 509.204,Z 555.792,A -85,B 0,C 180,E1 -5489.209,E2 -5489.209} C_VEL
LIN {X 0,Y 509.21,Z 556.018,A -85,B 0,C 180,E1 -5490,E2 -5490} C_VEL
LIN {X 0,Y 509.203,Z 555.799,A -85,B 0,C 180,E1 -5490.79,E2 -5490.79} C_VEL
LIN {X 0,Y 509.245,Z 554.171,A -85,B 0,C 180,E1 -5492.372,E2 -5492.372} C_VEL
LIN {X 0,Y 509.306,Z 552.753,A -85,B 0,C 180,E1 -5493.164,E2 -5493.164} C_VEL
LIN {X 0,Y 509.3,Z 549.755,A -85,B 0,C 180,E1 -5494.352,E2 -5494.352} C_VEL
LIN {X 0,Y 509.345,Z 545.702,A -85,B 0,C 180,E1 -5495.542,E2 -5495.542} C_VEL
LIN {X 0,Y 509.416,Z 539.828,A -85,B 0,C 180,E1 -5496.864,E2 -5496.864} C_VEL
LIN {X 0,Y 509.502,Z 532.667,A -85,B 0,C 180,E1 -5498.128,E2 -5498.128} C_VEL
LIN {X 0,Y 509.687,Z 524.246,A -85,B 0,C 180,E1 -5499.324,E2 -5499.324} C_VEL
LIN {X 0,Y 509.935,Z 515.628,A -85,B 0,C 180,E1 -5500.321,E2 -5500.321} C_VEL
LIN {X 0,Y 510.25,Z 505.001,A -85,B 0,C 180,E1 -5501.319,E2 -5501.319} C_VEL
LIN {X 0,Y 510.559,Z 493.019,A -85,B 0,C 180,E1 -5502.221,E2 -5502.221} C_VEL
LIN {X 0,Y 510.868,Z 481.069,A -85,B 0,C 180,E1 -5502.917,E2 -5502.917} C_VEL
LIN {X 0,Y 511.239,Z 468.636,A -85,B 0,C 180,E1 -5503.464,E2 -5503.464} C_VEL
LIN {X 0,Y 511.548,Z 455.894,A -85,B 0,C 180,E1 -5503.86,E2 -5503.86} C_VEL
LIN {X 0,Y 511.746,Z 442.586,A -85,B 0,C 180,E1 -5504.108,E2 -5504.108} C_VEL
LIN {X 0,Y 511.99,Z 354.301,A -85,B 0,C 180,E1 -5505.353,E2 -5505.353} C_VEL
LIN {X 0,Y 510.381,Z 340.453,A -85,B 0,C 180,E1 -5505.607,E2 -5505.607} C_VEL
LIN {X 0,Y 510.414,Z 333.716,A -85,B 0,C 180,E1 -5506.395,E2 -5506.395} C_VEL
LIN {X 0,Y 510.864,Z 312.071,A -85,B 0,C 180,E1 -5509.07,E2 -5509.07} C_VEL
LIN {X 0,Y 511.396,Z 286.909,A -85,B 0,C 180,E1 -5512.204,E2 -5512.204} C_VEL
LIN {X 0,Y 511.796,Z 267.079,A -85,B 0,C 180,E1 -5514.698,E2 -5514.698} C_VEL
LIN {X 0,Y 512.081,Z 253.317,A -85,B 0,C 180,E1 -5516.446,E2 -5516.446} C_VEL
LIN {X 0,Y 509.804,Z 242.133,A -85,B 0,C 180,E1 -5518,E2 -5518} C_VEL
LIN {X 0,Y 509.81,Z 241.982,A -85,B 0,C 180,E1 -5521.273,E2 -5521.273} C_VEL
LIN {X 0,Y 509.827,Z 241.976,A -85,B 0,C 180,E1 -5524.414,E2 -5524.414} C_VEL
LIN {X 0,Y 509.758,Z 241.991,A -85,B 0,C 180,E1 -5527.344,E2 -5527.344} C_VEL
LIN {X 0,Y 509.785,Z 241.979,A -85,B 0,C 180,E1 -5530.386,E2 -5530.386} C_VEL
LIN {X 0,Y 509.782,Z 241.984,A -85,B 0,C 180,E1 -5533.574,E2 -5533.574} C_VEL
LIN {X 0,Y 509.783,Z 241.979,A -85,B 0,C 180,E1 -5536.424,E2 -5536.424} C_VEL
LIN {X 0,Y 509.803,Z 241.979,A -85,B 0,C 180,E1 -5539.614,E2 -5539.614} C_VEL
LIN {X 0,Y 509.771,Z 241.983,A -85,B 0,C 180,E1 -5542.655,E2 -5542.655} C_VEL
LIN {X 0,Y 509.82,Z 241.975,A -85,B 0,C 180,E1 -5545.801,E2 -5545.801} C_VEL
LIN {X 0,Y 509.803,Z 241.981,A -85,B 0,C 180,E1 -5548.725,E2 -5548.725} C_VEL
LIN {X 0,Y 509.818,Z 241.981,A -85,B 0,C 180,E1 -5551.152,E2 -5551.152} C_VEL
LIN {X 0,Y 509.816,Z 241.975,A -85,B 0,C 180,E1 -5553.824,E2 -5553.824} C_VEL
LIN {X 0,Y 509.798,Z 241.98,A -85,B 0,C 180,E1 -5556.435,E2 -5556.435} C_VEL
LIN {X 0,Y 509.876,Z 241.967,A -85,B 0,C 180,E1 -5559.843,E2 -5559.843} C_VEL
LIN {X 0,Y 509.831,Z 241.977,A -85,B 0,C 180,E1 -5563.173,E2 -5563.173} C_VEL
LIN {X 0,Y 509.827,Z 241.974,A -85,B 0,C 180,E1 -5565.633,E2 -5565.633} C_VEL
LIN {X 0,Y 509.892,Z 241.972,A -85,B 0,C 180,E1 -5568.874,E2 -5568.874} C_VEL
LIN {X 0,Y 509.864,Z 241.971,A -85,B 0,C 180,E1 -5572.077,E2 -5572.077} C_VEL
LIN {X 0,Y 509.917,Z 241.969,A -85,B 0,C 180,E1 -5574.464,E2 -5574.464} C_VEL
LIN {X 0,Y 510.026,Z 241.949,A -85,B 0,C 180,E1 -5577.631,E2 -5577.631} C_VEL
LIN {X 0,Y 510.023,Z 241.954,A -85,B 0,C 180,E1 -5580.79,E2 -5580.79} C_VEL
LIN {X 0,Y 509.871,Z 241.969,A -85,B 0,C 180,E1 -5583.161,E2 -5583.161} C_VEL
LIN {X 0,Y 509.902,Z 241.972,A -85,B 0,C 180,E1 -5586.331,E2 -5586.331} C_VEL
LIN {X 0,Y 509.83,Z 241.973,A -85,B 0,C 180,E1 -5589.522,E2 -5589.522} C_VEL
LIN {X 0,Y 509.887,Z 241.97,A -85,B 0,C 180,E1 -5591.932,E2 -5591.932} C_VEL
LIN {X 0,Y 509.882,Z 241.967,A -85,B 0,C 180,E1 -5595.242,E2 -5595.242} C_VEL
LIN {X 0,Y 509.821,Z 241.979,A -85,B 0,C 180,E1 -5598.486,E2 -5598.486} C_VEL
LIN {X 0,Y 509.83,Z 241.973,A -85,B 0,C 180,E1 -5601.003,E2 -5601.003} C_VEL
LIN {X 0,Y 509.806,Z 241.978,A -85,B 0,C 180,E1 -5603.565,E2 -5603.565} C_VEL
LIN {X 0,Y 509.794,Z 241.982,A -85,B 0,C 180,E1 -5606.355,E2 -5606.355} C_VEL
LIN {X 0,Y 509.822,Z 241.975,A -85,B 0,C 180,E1 -5608.848,E2 -5608.848} C_VEL
LIN {X 0,Y 509.792,Z 241.981,A -85,B 0,C 180,E1 -5611.593,E2 -5611.593} C_VEL
LIN {X 0,Y 509.823,Z 241.977,A -85,B 0,C 180,E1 -5614.416,E2 -5614.416} C_VEL
LIN {X 0,Y 509.767,Z 241.983,A -85,B 0,C 180,E1 -5617.346,E2 -5617.346} C_VEL
LIN {X 0,Y 509.778,Z 241.982,A -85,B 0,C 180,E1 -5620.389,E2 -5620.389} C_VEL
LIN {X 0,Y 509.784,Z 241.985,A -85,B 0,C 180,E1 -5623.576,E2 -5623.576} C_VEL
LIN {X 0,Y 509.786,Z 241.98,A -85,B 0,C 180,E1 -5626.426,E2 -5626.426} C_VEL
LIN {X 0,Y 509.782,Z 241.987,A -85,B 0,C 180,E1 -5629.614,E2 -5629.614} C_VEL
LIN {X 0,Y 509.773,Z 241.98,A -85,B 0,C 180,E1 -5632.657,E2 -5632.657} C_VEL
LIN {X 0,Y 509.756,Z 241.99,A -85,B 0,C 180,E1 -5633.738,E2 -5633.738} C_VEL
LIN {X 0,Y 509.094,Z 242.068,A -85,B 0,C 180,E1 -5634.398,E2 -5634.398} C_VEL
LIN {X 0,Y 506.272,Z 242.424,A -85,B 0,C 180,E1 -5635.47,E2 -5635.47} C_VEL
LIN {X 0,Y 503.88,Z 242.719,A -85,B 0,C 180,E1 -5636.334,E2 -5636.334} C_VEL
LIN {X 0,Y 502.842,Z 242.845,A -85,B 0,C 180,E1 -5637.001,E2 -5637.001} C_VEL
LIN {X 0,Y 502.752,Z 242.856,A -85,B 0,C 180,E1 -5637.227,E2 -5637.227} C_VEL
LIN {X 0,Y 502.745,Z 242.858,A -85,B 0,C 180,E1 -5640.08,E2 -5640.08} C_VEL
LIN {X 0,Y 502.767,Z 242.853,A -85,B 0,C 180,E1 -5642.53,E2 -5642.53} C_VEL
LIN {X 0,Y 502.762,Z 242.861,A -85,B 0,C 180,E1 -5645.317,E2 -5645.317} C_VEL
LIN {X 0,Y 502.773,Z 242.855,A -85,B 0,C 180,E1 -5647.827,E2 -5647.827} C_VEL
LIN {X 0,Y 502.777,Z 242.852,A -85,B 0,C 180,E1 -5650.399,E2 -5650.399} C_VEL
LIN {X 0,Y 502.792,Z 242.854,A -85,B 0,C 180,E1 -5652.931,E2 -5652.931} C_VEL
LIN {X 0,Y 502.797,Z 242.856,A -85,B 0,C 180,E1 -5655.428,E2 -5655.428} C_VEL
LIN {X 0,Y 502.841,Z 242.848,A -85,B 0,C 180,E1 -5658.717,E2 -5658.717} C_VEL
LIN {X 0,Y 502.869,Z 242.918,A -85,B 0,C 180,E1 -5662.345,E2 -5662.345} C_VEL
LIN {X 0,Y 503.019,Z 243.726,A -85,B 0,C 180,E1 -5662.503,E2 -5662.503} C_VEL
LIN {X 0,Y 505.416,Z 250.773,A -85,B 0,C 180,E1 -5662.707,E2 -5662.707} C_VEL
LIN {X 0,Y 505.058,Z 331.766,A -85,B 0,C 180,E1 -5663.885,E2 -5663.885} C_VEL
LIN {X 0,Y 504.942,Z 344.679,A -85,B 0,C 180,E1 -5664.234,E2 -5664.234} C_VEL
LIN {X 0,Y 504.766,Z 357.668,A -85,B 0,C 180,E1 -5664.758,E2 -5664.758} C_VEL
LIN {X 0,Y 504.483,Z 369.418,A -85,B 0,C 180,E1 -5665.406,E2 -5665.406} C_VEL
LIN {X 0,Y 504.166,Z 380.64,A -85,B 0,C 180,E1 -5666.204,E2 -5666.204} C_VEL
LIN {X 0,Y 503.79,Z 390.779,A -85,B 0,C 180,E1 -5667.102,E2 -5667.102} C_VEL
LIN {X 0,Y 503.558,Z 399.054,A -85,B 0,C 180,E1 -5668.001,E2 -5668.001} C_VEL
LIN {X 0,Y 503.273,Z 406.717,A -85,B 0,C 180,E1 -5669,E2 -5669} C_VEL
LIN {X 0,Y 502.955,Z 414.224,A -85,B 0,C 180,E1 -5670.2,E2 -5670.2} C_VEL
LIN {X 0,Y 502.671,Z 421.14,A -85,B 0,C 180,E1 -5671.603,E2 -5671.603} C_VEL
LIN {X 0,Y 502.539,Z 425.746,A -85,B 0,C 180,E1 -5672.806,E2 -5672.806} C_VEL
LIN {X 0,Y 502.468,Z 429.275,A -85,B 0,C 180,E1 -5674.01,E2 -5674.01} C_VEL
LIN {X 0,Y 502.509,Z 431.091,A -85,B 0,C 180,E1 -5674.814,E2 -5674.814} C_VEL
LIN {X 0,Y 502.405,Z 433.454,A -85,B 0,C 180,E1 -5676.426,E2 -5676.426} C_VEL
LIN {X 0,Y 502.418,Z 434.055,A -85,B 0,C 180,E1 -5677.233,E2 -5677.233} C_VEL
LIN {X 0,Y 502.356,Z 434.284,A -85,B 0,C 180,E1 -5678.042,E2 -5678.042} C_VEL
LIN {X 0,Y 502.365,Z 434.075,A -85,B 0,C 180,E1 -5678.852,E2 -5678.852} C_VEL
LIN {X 0,Y 502.363,Z 432.505,A -85,B 0,C 180,E1 -5680.479,E2 -5680.479} C_VEL
LIN {X 0,Y 502.505,Z 430.106,A -85,B 0,C 180,E1 -5681.756,E2 -5681.756} C_VEL
LIN {X 0,Y 502.582,Z 426.954,A -85,B 0,C 180,E1 -5682.929,E2 -5682.929} C_VEL
LIN {X 0,Y 502.69,Z 422.581,A -85,B 0,C 180,E1 -5684.162,E2 -5684.162} C_VEL
LIN {X 0,Y 502.932,Z 416.963,A -85,B 0,C 180,E1 -5685.397,E2 -5685.397} C_VEL
LIN {X 0,Y 503.174,Z 409.842,A -85,B 0,C 180,E1 -5686.638,E2 -5686.638} C_VEL
LIN {X 0,Y 503.463,Z 400.881,A -85,B 0,C 180,E1 -5687.885,E2 -5687.885} C_VEL
LIN {X 0,Y 503.812,Z 391.589,A -85,B 0,C 180,E1 -5688.925,E2 -5688.925} C_VEL
LIN {X 0,Y 504.124,Z 381.112,A -85,B 0,C 180,E1 -5689.865,E2 -5689.865} C_VEL
LIN {X 0,Y 504.488,Z 370.398,A -85,B 0,C 180,E1 -5690.634,E2 -5690.634} C_VEL
LIN {X 0,Y 504.773,Z 359.052,A -85,B 0,C 180,E1 -5691.276,E2 -5691.276} C_VEL
LIN {X 0,Y 504.938,Z 346.521,A -85,B 0,C 180,E1 -5691.805,E2 -5691.805} C_VEL
LIN {X 0,Y 505.107,Z 333.524,A -85,B 0,C 180,E1 -5692.173,E2 -5692.173} C_VEL
LIN {X 0,Y 505.184,Z 309.917,A -85,B 0,C 180,E1 -5692.547,E2 -5692.547} C_VEL
LIN {X 0,Y 505.424,Z 250.749,A -85,B 0,C 180,E1 -5693.401,E2 -5693.401} C_VEL
LIN {X 0,Y 502.975,Z 243.716,A -85,B 0,C 180,E1 -5693.613,E2 -5693.613} C_VEL
LIN {X 0,Y 502.818,Z 242.939,A -85,B 0,C 180,E1 -5693.763,E2 -5693.763} C_VEL
LIN {X 0,Y 502.786,Z 242.856,A -85,B 0,C 180,E1 -5696.57,E2 -5696.57} C_VEL
LIN {X 0,Y 502.816,Z 242.848,A -85,B 0,C 180,E1 -5699.934,E2 -5699.934} C_VEL
LIN {X 0,Y 502.804,Z 242.856,A -85,B 0,C 180,E1 -5703.033,E2 -5703.033} C_VEL
LIN {X 0,Y 502.765,Z 242.844,A -85,B 0,C 180,E1 -5705.951,E2 -5705.951} C_VEL
LIN {X 0,Y 502.782,Z 242.857,A -85,B 0,C 180,E1 -5708.977,E2 -5708.977} C_VEL
LIN {X 0,Y 502.77,Z 242.853,A -85,B 0,C 180,E1 -5712.194,E2 -5712.194} C_VEL
LIN {X 0,Y 502.783,Z 242.851,A -85,B 0,C 180,E1 -5715.469,E2 -5715.469} C_VEL
LIN {X 0,Y 502.761,Z 242.858,A -85,B 0,C 180,E1 -5718.928,E2 -5718.928} C_VEL
LIN {X 0,Y 502.757,Z 242.854,A -85,B 0,C 180,E1 -5722.042,E2 -5722.042} C_VEL
LIN {X 0,Y 502.786,Z 242.853,A -85,B 0,C 180,E1 -5725.033,E2 -5725.033} C_VEL
LIN {X 0,Y 502.778,Z 242.855,A -85,B 0,C 180,E1 -5727.915,E2 -5727.915} C_VEL
LIN {X 0,Y 502.807,Z 242.847,A -85,B 0,C 180,E1 -5730.711,E2 -5730.711} C_VEL
LIN {X 0,Y 502.77,Z 242.855,A -85,B 0,C 180,E1 -5733.459,E2 -5733.459} C_VEL
LIN {X 0,Y 502.766,Z 242.854,A -85,B 0,C 180,E1 -5736.085,E2 -5736.085} C_VEL
LIN {X 0,Y 502.774,Z 242.842,A -85,B 0,C 180,E1 -5738.688,E2 -5738.688} C_VEL
LIN {X 0,Y 502.815,Z 242.846,A -85,B 0,C 180,E1 -5741.247,E2 -5741.247} C_VEL
LIN {X 0,Y 502.842,Z 242.842,A -85,B 0,C 180,E1 -5744.6,E2 -5744.6} C_VEL
LIN {X 0,Y 502.87,Z 242.847,A -85,B 0,C 180,E1 -5748.039,E2 -5748.039} C_VEL
LIN {X 0,Y 502.84,Z 242.84,A -85,B 0,C 180,E1 -5751.156,E2 -5751.156} C_VEL
LIN {X 0,Y 502.861,Z 242.847,A -85,B 0,C 180,E1 -5753.58,E2 -5753.58} C_VEL
LIN {X 0,Y 502.826,Z 242.843,A -85,B 0,C 180,E1 -5756.795,E2 -5756.795} C_VEL
LIN {X 0,Y 502.882,Z 242.84,A -85,B 0,C 180,E1 -5758.398,E2 -5758.398} C_VEL
LIN {X 0,Y 502.991,Z 242.828,A -85,B 0,C 180,E1 -5760,E2 -5760} C_VEL
LIN {X 0,Y 503.004,Z 242.821,A -85,B 0,C 180,E1 -5762.402,E2 -5762.402} C_VEL
LIN {X 0,Y 502.879,Z 242.845,A -85,B 0,C 180,E1 -5765.614,E2 -5765.614} C_VEL
LIN {X 0,Y 502.862,Z 242.841,A -85,B 0,C 180,E1 -5768.034,E2 -5768.034} C_VEL
LIN {X 0,Y 502.864,Z 242.848,A -85,B 0,C 180,E1 -5771.283,E2 -5771.283} C_VEL
LIN {X 0,Y 502.815,Z 242.847,A -85,B 0,C 180,E1 -5774.572,E2 -5774.572} C_VEL
LIN {X 0,Y 502.808,Z 242.848,A -85,B 0,C 180,E1 -5777.909,E2 -5777.909} C_VEL
LIN {X 0,Y 502.822,Z 242.848,A -85,B 0,C 180,E1 -5780.536,E2 -5780.536} C_VEL
LIN {X 0,Y 502.778,Z 242.856,A -85,B 0,C 180,E1 -5783.041,E2 -5783.041} C_VEL
LIN {X 0,Y 502.768,Z 242.852,A -85,B 0,C 180,E1 -5785.68,E2 -5785.68} C_VEL
LIN {X 0,Y 502.762,Z 242.848,A -85,B 0,C 180,E1 -5788.377,E2 -5788.377} C_VEL
LIN {X 0,Y 502.758,Z 242.862,A -85,B 0,C 180,E1 -5791.146,E2 -5791.146} C_VEL
LIN {X 0,Y 502.779,Z 242.846,A -85,B 0,C 180,E1 -5793.996,E2 -5793.996} C_VEL
LIN {X 0,Y 502.731,Z 242.862,A -85,B 0,C 180,E1 -5797.172,E2 -5797.172} C_VEL
LIN {X 0,Y 502.765,Z 242.854,A -85,B 0,C 180,E1 -5800.017,E2 -5800.017} C_VEL
LIN {X 0,Y 502.734,Z 242.86,A -85,B 0,C 180,E1 -5803.236,E2 -5803.236} C_VEL
LIN {X 0,Y 502.762,Z 242.854,A -85,B 0,C 180,E1 -5805.659,E2 -5805.659} C_VEL
LIN {X 0,Y 502.754,Z 242.858,A -85,B 0,C 180,E1 -5808.928,E2 -5808.928} C_VEL
LIN {X 0,Y 502.743,Z 242.856,A -85,B 0,C 180,E1 -5812.042,E2 -5812.042} C_VEL
LIN {X 0,Y 502.779,Z 242.851,A -85,B 0,C 180,E1 -5815.033,E2 -5815.033} C_VEL
LIN {X 0,Y 502.756,Z 242.855,A -85,B 0,C 180,E1 -5817.914,E2 -5817.914} C_VEL
LIN {X 0,Y 502.748,Z 242.859,A -85,B 0,C 180,E1 -5820.708,E2 -5820.708} C_VEL
LIN {X 0,Y 502.783,Z 243.112,A -85,B 0,C 180,E1 -5821.783,E2 -5821.783} C_VEL
LIN {X 0,Y 505.1,Z 254.229,A -85,B 0,C 180,E1 -5823.384,E2 -5823.384} C_VEL
LIN {X 0,Y 504.982,Z 264.232,A -85,B 0,C 180,E1 -5824.693,E2 -5824.693} C_VEL
LIN {X 0,Y 504.397,Z 287.519,A -85,B 0,C 180,E1 -5827.686,E2 -5827.686} C_VEL
LIN {X 0,Y 503.817,Z 310.955,A -85,B 0,C 180,E1 -5830.652,E2 -5830.652} C_VEL
LIN {X 0,Y 503.341,Z 334.32,A -85,B 0,C 180,E1 -5833.576,E2 -5833.576} C_VEL
LIN {X 0,Y 503.311,Z 339.084,A -85,B 0,C 180,E1 -5834.151,E2 -5834.151} C_VEL
LIN {X 0,Y 505.267,Z 357.533,A -85,B 0,C 180,E1 -5834.499,E2 -5834.499} C_VEL
LIN {X 0,Y 504.774,Z 449.224,A -85,B 0,C 180,E1 -5835.821,E2 -5835.821} C_VEL
LIN {X 0,Y 504.398,Z 462.6,A -85,B 0,C 180,E1 -5836.17,E2 -5836.17} C_VEL
LIN {X 0,Y 504.115,Z 476.017,A -85,B 0,C 180,E1 -5836.701,E2 -5836.701} C_VEL
LIN {X 0,Y 503.68,Z 488.545,A -85,B 0,C 180,E1 -5837.385,E2 -5837.385} C_VEL
LIN {X 0,Y 503.367,Z 500.344,A -85,B 0,C 180,E1 -5838.218,E2 -5838.218} C_VEL
LIN {X 0,Y 503.027,Z 510.688,A -85,B 0,C 180,E1 -5839.128,E2 -5839.128} C_VEL
LIN {X 0,Y 502.721,Z 520.01,A -85,B 0,C 180,E1 -5840.139,E2 -5840.139} C_VEL
LIN {X 0,Y 502.484,Z 529.112,A -85,B 0,C 180,E1 -5841.352,E2 -5841.352} C_VEL
LIN {X 0,Y 502.353,Z 536.459,A -85,B 0,C 180,E1 -5842.564,E2 -5842.564} C_VEL
LIN {X 0,Y 502.235,Z 541.419,A -85,B 0,C 180,E1 -5843.572,E2 -5843.572} C_VEL
LIN {X 0,Y 502.214,Z 546.255,A -85,B 0,C 180,E1 -5844.781,E2 -5844.781} C_VEL
LIN {X 0,Y 502.264,Z 549.961,A -85,B 0,C 180,E1 -5845.988,E2 -5845.988} C_VEL
LIN {X 0,Y 502.251,Z 551.87,A -85,B 0,C 180,E1 -5846.791,E2 -5846.791} C_VEL
LIN {X 0,Y 502.191,Z 553.296,A -85,B 0,C 180,E1 -5847.594,E2 -5847.594} C_VEL
LIN {X 0,Y 502.153,Z 554.943,A -85,B 0,C 180,E1 -5849.198,E2 -5849.198} C_VEL
LIN {X 0,Y 502.161,Z 555.17,A -85,B 0,C 180,E1 -5850,E2 -5850} C_VEL
LIN {X 0,Y 502.152,Z 554.951,A -85,B 0,C 180,E1 -5850.802,E2 -5850.802} C_VEL
LIN {X 0,Y 502.189,Z 553.324,A -85,B 0,C 180,E1 -5852.406,E2 -5852.406} C_VEL
LIN {X 0,Y 502.25,Z 551.906,A -85,B 0,C 180,E1 -5853.208,E2 -5853.208} C_VEL
LIN {X 0,Y 502.233,Z 548.906,A -85,B 0,C 180,E1 -5854.414,E2 -5854.414} C_VEL
LIN {X 0,Y 502.282,Z 544.853,A -85,B 0,C 180,E1 -5855.62,E2 -5855.62} C_VEL
LIN {X 0,Y 502.335,Z 538.72,A -85,B 0,C 180,E1 -5857.011,E2 -5857.011} C_VEL
LIN {X 0,Y 502.438,Z 531.814,A -85,B 0,C 180,E1 -5858.243,E2 -5858.243} C_VEL
LIN {X 0,Y 502.602,Z 523.388,A -85,B 0,C 180,E1 -5859.456,E2 -5859.456} C_VEL
LIN {X 0,Y 502.861,Z 514.769,A -85,B 0,C 180,E1 -5860.468,E2 -5860.468} C_VEL
LIN {X 0,Y 503.169,Z 504.138,A -85,B 0,C 180,E1 -5861.48,E2 -5861.48} C_VEL
LIN {X 0,Y 503.537,Z 493.359,A -85,B 0,C 180,E1 -5862.309,E2 -5862.309} C_VEL
LIN {X 0,Y 503.851,Z 482.16,A -85,B 0,C 180,E1 -5862.998,E2 -5862.998} C_VEL
LIN {X 0,Y 504.248,Z 470.396,A -85,B 0,C 180,E1 -5863.551,E2 -5863.551} C_VEL
LIN {X 0,Y 504.594,Z 456.871,A -85,B 0,C 180,E1 -5864.004,E2 -5864.004} C_VEL
LIN {X 0,Y 504.853,Z 443.504,A -85,B 0,C 180,E1 -5864.279,E2 -5864.279} C_VEL
LIN {X 0,Y 505.154,Z 355.355,A -85,B 0,C 180,E1 -5865.539,E2 -5865.539} C_VEL
LIN {X 0,Y 503.31,Z 339.42,A -85,B 0,C 180,E1 -5865.84,E2 -5865.84} C_VEL
LIN {X 0,Y 503.815,Z 314.535,A -85,B 0,C 180,E1 -5868.924,E2 -5868.924} C_VEL
LIN {X 0,Y 504.375,Z 289.352,A -85,B 0,C 180,E1 -5872.099,E2 -5872.099} C_VEL
LIN {X 0,Y 504.809,Z 270.736,A -85,B 0,C 180,E1 -5874.467,E2 -5874.467} C_VEL
LIN {X 0,Y 505.161,Z 255.386,A -85,B 0,C 180,E1 -5876.435,E2 -5876.435} C_VEL
LIN {X 0,Y 503.502,Z 246.528,A -85,B 0,C 180,E1 -5877.652,E2 -5877.652} C_VEL
LIN {X 0,Y 502.759,Z 242.965,A -85,B 0,C 180,E1 -5878.195,E2 -5878.195} C_VEL
LIN {X 0,Y 502.761,Z 242.861,A -85,B 0,C 180,E1 -5881.492,E2 -5881.492} C_VEL
LIN {X 0,Y 502.779,Z 242.854,A -85,B 0,C 180,E1 -5884.44,E2 -5884.44} C_VEL
LIN {X 0,Y 502.716,Z 242.865,A -85,B 0,C 180,E1 -5887.168,E2 -5887.168} C_VEL
LIN {X 0,Y 502.728,Z 242.859,A -85,B 0,C 180,E1 -5890.019,E2 -5890.019} C_VEL
LIN {X 0,Y 502.737,Z 242.857,A -85,B 0,C 180,E1 -5892.191,E2 -5892.191} C_VEL
LIN {X 0,Y 502.769,Z 242.858,A -85,B 0,C 180,E1 -5895.47,E2 -5895.47} C_VEL
LIN {X 0,Y 502.752,Z 242.86,A -85,B 0,C 180,E1 -5898.927,E2 -5898.927} C_VEL
LIN {X 0,Y 502.75,Z 242.855,A -85,B 0,C 180,E1 -5902.042,E2 -5902.042} C_VEL
LIN {X 0,Y 502.77,Z 242.861,A -85,B 0,C 180,E1 -5905.032,E2 -5905.032} C_VEL
LIN {X 0,Y 502.744,Z 242.856,A -85,B 0,C 180,E1 -5907.913,E2 -5907.913} C_VEL
LIN {X 0,Y 502.777,Z 242.857,A -85,B 0,C 180,E1 -5910.709,E2 -5910.709} C_VEL
LIN {X 0,Y 502.758,Z 242.856,A -85,B 0,C 180,E1 -5913.46,E2 -5913.46} C_VEL
LIN {X 0,Y 502.743,Z 242.856,A -85,B 0,C 180,E1 -5916.084,E2 -5916.084} C_VEL
LIN {X 0,Y 502.76,Z 242.86,A -85,B 0,C 180,E1 -5918.688,E2 -5918.688} C_VEL
LIN {X 0,Y 502.792,Z 242.853,A -85,B 0,C 180,E1 -5921.247,E2 -5921.247} C_VEL
LIN {X 0,Y 502.821,Z 242.854,A -85,B 0,C 180,E1 -5924.664,E2 -5924.664} C_VEL
LIN {X 0,Y 502.863,Z 242.842,A -85,B 0,C 180,E1 -5928.039,E2 -5928.039} C_VEL
LIN {X 0,Y 502.826,Z 242.848,A -85,B 0,C 180,E1 -5931.156,E2 -5931.156} C_VEL
LIN {X 0,Y 502.833,Z 242.845,A -85,B 0,C 180,E1 -5933.58,E2 -5933.58} C_VEL
LIN {X 0,Y 502.848,Z 242.848,A -85,B 0,C 180,E1 -5936.795,E2 -5936.795} C_VEL
LIN {X 0,Y 502.884,Z 242.845,A -85,B 0,C 180,E1 -5938.398,E2 -5938.398} C_VEL
LIN {X 0,Y 502.974,Z 242.832,A -85,B 0,C 180,E1 -5940.801,E2 -5940.801} C_VEL
LIN {X 0,Y 502.99,Z 242.833,A -85,B 0,C 180,E1 -5942.403,E2 -5942.403} C_VEL
LIN {X 0,Y 502.88,Z 242.839,A -85,B 0,C 180,E1 -5945.614,E2 -5945.614} C_VEL
LIN {X 0,Y 502.831,Z 242.849,A -85,B 0,C 180,E1 -5948.035,E2 -5948.035} C_VEL
LIN {X 0,Y 502.821,Z 242.846,A -85,B 0,C 180,E1 -5951.285,E2 -5951.285} C_VEL
LIN {X 0,Y 502.82,Z 242.851,A -85,B 0,C 180,E1 -5954.572,E2 -5954.572} C_VEL
LIN {X 0,Y 502.787,Z 242.855,A -85,B 0,C 180,E1 -5957.91,E2 -5957.91} C_VEL
LIN {X 0,Y 502.818,Z 242.85,A -85,B 0,C 180,E1 -5960.537,E2 -5960.537} C_VEL
LIN {X 0,Y 502.775,Z 242.852,A -85,B 0,C 180,E1 -5963.042,E2 -5963.042} C_VEL
LIN {X 0,Y 502.758,Z 242.858,A -85,B 0,C 180,E1 -5965.68,E2 -5965.68} C_VEL
LIN {X 0,Y 502.758,Z 242.858,A -85,B 0,C 180,E1 -5968.378,E2 -5968.378} C_VEL
LIN {X 0,Y 502.775,Z 242.852,A -85,B 0,C 180,E1 -5971.145,E2 -5971.145} C_VEL
LIN {X 0,Y 502.774,Z 242.86,A -85,B 0,C 180,E1 -5973.997,E2 -5973.997} C_VEL
LIN {X 0,Y 502.721,Z 242.86,A -85,B 0,C 180,E1 -5977.171,E2 -5977.171} C_VEL
LIN {X 0,Y 502.722,Z 242.865,A -85,B 0,C 180,E1 -5980.022,E2 -5980.022} C_VEL
LIN {X 0,Y 502.729,Z 242.86,A -85,B 0,C 180,E1 -5983.237,E2 -5983.237} C_VEL
LIN {X 0,Y 502.762,Z 242.861,A -85,B 0,C 180,E1 -5985.66,E2 -5985.66} C_VEL
LIN {X 0,Y 502.746,Z 242.857,A -85,B 0,C 180,E1 -5989.015,E2 -5989.015} C_VEL
LIN {X 0,Y 502.752,Z 242.858,A -85,B 0,C 180,E1 -5992.044,E2 -5992.044} C_VEL
LIN {X 0,Y 502.749,Z 242.857,A -85,B 0,C 180,E1 -5995.032,E2 -5995.032} C_VEL
LIN {X 0,Y 502.752,Z 242.856,A -85,B 0,C 180,E1 -5997.227,E2 -5997.227} C_VEL
LIN {X 0,Y 502.066,Z 242.945,A -85,B 0,C 180,E1 -5997.895,E2 -5997.895} C_VEL
LIN {X 0,Y 499.197,Z 243.3,A -85,B 0,C 180,E1 -5998.981,E2 -5998.981} C_VEL
LIN {X 0,Y 496.787,Z 243.602,A -85,B 0,C 180,E1 -5999.856,E2 -5999.856} C_VEL
LIN {X 0,Y 495.761,Z 243.726,A -85,B 0,C 180,E1 -6000.532,E2 -6000.532} C_VEL
LIN {X 0,Y 495.681,Z 243.736,A -85,B 0,C 180,E1 -6000.761,E2 -6000.761} C_VEL
LIN {X 0,Y 495.72,Z 243.737,A -85,B 0,C 180,E1 -6003.276,E2 -6003.276} C_VEL
LIN {X 0,Y 495.702,Z 243.738,A -85,B 0,C 180,E1 -6005.723,E2 -6005.723} C_VEL
LIN {X 0,Y 495.731,Z 243.73,A -85,B 0,C 180,E1 -6008.371,E2 -6008.371} C_VEL
LIN {X 0,Y 495.753,Z 243.731,A -85,B 0,C 180,E1 -6010.971,E2 -6010.971} C_VEL
LIN {X 0,Y 495.743,Z 243.733,A -85,B 0,C 180,E1 -6013.53,E2 -6013.53} C_VEL
LIN {X 0,Y 495.753,Z 243.727,A -85,B 0,C 180,E1 -6016.055,E2 -6016.055} C_VEL
LIN {X 0,Y 495.826,Z 243.72,A -85,B 0,C 180,E1 -6018.555,E2 -6018.555} C_VEL
LIN {X 0,Y 495.846,Z 243.91,A -85,B 0,C 180,E1 -6022.175,E2 -6022.175} C_VEL
LIN {X 0,Y 496.016,Z 244.801,A -85,B 0,C 180,E1 -6022.3,E2 -6022.3} C_VEL
LIN {X 0,Y 498.687,Z 252.927,A -85,B 0,C 180,E1 -6022.521,E2 -6022.521} C_VEL
LIN {X 0,Y 498.233,Z 332.814,A -85,B 0,C 180,E1 -6023.699,E2 -6023.699} C_VEL
LIN {X 0,Y 498.074,Z 345.685,A -85,B 0,C 180,E1 -6024.053,E2 -6024.053} C_VEL
LIN {X 0,Y 497.908,Z 358.631,A -85,B 0,C 180,E1 -6024.584,E2 -6024.584} C_VEL
LIN {X 0,Y 497.6,Z 370.354,A -85,B 0,C 180,E1 -6025.241,E2 -6025.241} C_VEL
LIN {X 0,Y 497.256,Z 381.567,A -85,B 0,C 180,E1 -6026.05,E2 -6026.05} C_VEL
LIN {X 0,Y 496.878,Z 391.691,A -85,B 0,C 180,E1 -6026.96,E2 -6026.96} C_VEL
LIN {X 0,Y 496.576,Z 400.801,A -85,B 0,C 180,E1 -6027.973,E2 -6027.973} C_VEL
LIN {X 0,Y 496.251,Z 409.616,A -85,B 0,C 180,E1 -6029.189,E2 -6029.189} C_VEL
LIN {X 0,Y 495.909,Z 416.749,A -85,B 0,C 180,E1 -6030.406,E2 -6030.406} C_VEL
LIN {X 0,Y 495.652,Z 422.468,A -85,B 0,C 180,E1 -6031.625,E2 -6031.625} C_VEL
LIN {X 0,Y 495.512,Z 426.973,A -85,B 0,C 180,E1 -6032.846,E2 -6032.846} C_VEL
LIN {X 0,Y 495.435,Z 430.408,A -85,B 0,C 180,E1 -6034.068,E2 -6034.068} C_VEL
LIN {X 0,Y 495.468,Z 432.144,A -85,B 0,C 180,E1 -6034.882,E2 -6034.882} C_VEL
LIN {X 0,Y 495.36,Z 434.411,A -85,B 0,C 180,E1 -6036.517,E2 -6036.517} C_VEL
LIN {X 0,Y 495.365,Z 434.969,A -85,B 0,C 180,E1 -6037.336,E2 -6037.336} C_VEL
LIN {X 0,Y 495.321,Z 435.115,A -85,B 0,C 180,E1 -6038.157,E2 -6038.157} C_VEL
LIN {X 0,Y 495.333,Z 434.222,A -85,B 0,C 180,E1 -6039.803,E2 -6039.803} C_VEL
LIN {X 0,Y 495.351,Z 433.198,A -85,B 0,C 180,E1 -6040.629,E2 -6040.629} C_VEL
LIN {X 0,Y 495.492,Z 430.875,A -85,B 0,C 180,E1 -6041.848,E2 -6041.848} C_VEL
LIN {X 0,Y 495.572,Z 427.467,A -85,B 0,C 180,E1 -6043.115,E2 -6043.115} C_VEL
LIN {X 0,Y 495.73,Z 422.988,A -85,B 0,C 180,E1 -6044.365,E2 -6044.365} C_VEL
LIN {X 0,Y 495.999,Z 416.113,A -85,B 0,C 180,E1 -6045.829,E2 -6045.829} C_VEL
LIN {X 0,Y 496.294,Z 408.596,A -85,B 0,C 180,E1 -6047.088,E2 -6047.088} C_VEL
LIN {X 0,Y 496.587,Z 400.849,A -85,B 0,C 180,E1 -6048.141,E2 -6048.141} C_VEL
LIN {X 0,Y 496.974,Z 391.29,A -85,B 0,C 180,E1 -6049.195,E2 -6049.195} C_VEL
LIN {X 0,Y 497.305,Z 380.575,A -85,B 0,C 180,E1 -6050.149,E2 -6050.149} C_VEL
LIN {X 0,Y 497.699,Z 370.133,A -85,B 0,C 180,E1 -6050.89,E2 -6050.89} C_VEL
LIN {X 0,Y 497.964,Z 358.736,A -85,B 0,C 180,E1 -6051.528,E2 -6051.528} C_VEL
LIN {X 0,Y 498.115,Z 345.656,A -85,B 0,C 180,E1 -6052.065,E2 -6052.065} C_VEL
LIN {X 0,Y 498.292,Z 333.043,A -85,B 0,C 180,E1 -6052.41,E2 -6052.41} C_VEL
LIN {X 0,Y 498.509,Z 289.286,A -85,B 0,C 180,E1 -6053.07,E2 -6053.07} C_VEL
LIN {X 0,Y 498.585,Z 252.037,A -85,B 0,C 180,E1 -6053.617,E2 -6053.617} C_VEL
LIN {X 0,Y 495.989,Z 244.851,A -85,B 0,C 180,E1 -6053.834,E2 -6053.834} C_VEL
LIN {X 0,Y 495.774,Z 243.847,A -85,B 0,C 180,E1 -6053.989,E2 -6053.989} C_VEL
LIN {X 0,Y 495.734,Z 243.737,A -85,B 0,C 180,E1 -6056.979,E2 -6056.979} C_VEL
LIN {X 0,Y 495.765,Z 243.726,A -85,B 0,C 180,E1 -6060.146,E2 -6060.146} C_VEL
LIN {X 0,Y 495.753,Z 243.732,A -85,B 0,C 180,E1 -6063.236,E2 -6063.236} C_VEL
LIN {X 0,Y 495.708,Z 243.721,A -85,B 0,C 180,E1 -6066.086,E2 -6066.086} C_VEL
LIN {X 0,Y 495.74,Z 243.732,A -85,B 0,C 180,E1 -6068.764,E2 -6068.764} C_VEL
LIN {X 0,Y 495.724,Z 243.729,A -85,B 0,C 180,E1 -6071.784,E2 -6071.784} C_VEL
LIN {X 0,Y 495.736,Z 243.731,A -85,B 0,C 180,E1 -6075.14,E2 -6075.14} C_VEL
LIN {X 0,Y 495.721,Z 243.732,A -85,B 0,C 180,E1 -6078.215,E2 -6078.215} C_VEL
LIN {X 0,Y 495.737,Z 243.726,A -85,B 0,C 180,E1 -6081.235,E2 -6081.235} C_VEL
LIN {X 0,Y 495.732,Z 243.735,A -85,B 0,C 180,E1 -6084.46,E2 -6084.46} C_VEL
LIN {X 0,Y 495.763,Z 243.725,A -85,B 0,C 180,E1 -6087.405,E2 -6087.405} C_VEL
LIN {X 0,Y 495.758,Z 243.721,A -85,B 0,C 180,E1 -6090.253,E2 -6090.253} C_VEL
LIN {X 0,Y 495.735,Z 243.731,A -85,B 0,C 180,E1 -6093.27,E2 -6093.27} C_VEL
LIN {X 0,Y 495.714,Z 243.735,A -85,B 0,C 180,E1 -6095.723,E2 -6095.723} C_VEL
LIN {X 0,Y 495.734,Z 243.719,A -85,B 0,C 180,E1 -6098.37,E2 -6098.37} C_VEL
LIN {X 0,Y 495.771,Z 243.722,A -85,B 0,C 180,E1 -6100.971,E2 -6100.971} C_VEL
LIN {X 0,Y 495.817,Z 243.718,A -85,B 0,C 180,E1 -6104.548,E2 -6104.548} C_VEL
LIN {X 0,Y 495.821,Z 243.726,A -85,B 0,C 180,E1 -6107.965,E2 -6107.965} C_VEL
LIN {X 0,Y 495.798,Z 243.717,A -85,B 0,C 180,E1 -6111.029,E2 -6111.029} C_VEL
LIN {X 0,Y 495.812,Z 243.724,A -85,B 0,C 180,E1 -6113.489,E2 -6113.489} C_VEL
LIN {X 0,Y 495.695,Z 243.736,A -85,B 0,C 180,E1 -6115.935,E2 -6115.935} C_VEL
LIN {X 0,Y 495.966,Z 243.703,A -85,B 0,C 180,E1 -6117.563,E2 -6117.563} C_VEL
LIN {X 0,Y 495.961,Z 243.704,A -85,B 0,C 180,E1 -6120,E2 -6120} C_VEL
LIN {X 0,Y 495.972,Z 243.697,A -85,B 0,C 180,E1 -6122.436,E2 -6122.436} C_VEL
LIN {X 0,Y 495.836,Z 243.721,A -85,B 0,C 180,E1 -6125.694,E2 -6125.694} C_VEL
LIN {X 0,Y 495.821,Z 243.717,A -85,B 0,C 180,E1 -6128.149,E2 -6128.149} C_VEL
LIN {X 0,Y 495.84,Z 243.722,A -85,B 0,C 180,E1 -6131.445,E2 -6131.445} C_VEL
LIN {X 0,Y 495.766,Z 243.726,A -85,B 0,C 180,E1 -6134.783,E2 -6134.783} C_VEL
LIN {X 0,Y 495.772,Z 243.723,A -85,B 0,C 180,E1 -6138.172,E2 -6138.172} C_VEL
LIN {X 0,Y 495.767,Z 243.728,A -85,B 0,C 180,E1 -6140.757,E2 -6140.757} C_VEL
LIN {X 0,Y 495.73,Z 243.737,A -85,B 0,C 180,E1 -6143.388,E2 -6143.388} C_VEL
LIN {X 0,Y 495.731,Z 243.73,A -85,B 0,C 180,E1 -6146.73,E2 -6146.73} C_VEL
LIN {X 0,Y 495.732,Z 243.731,A -85,B 0,C 180,E1 -6149.749,E2 -6149.749} C_VEL
LIN {X 0,Y 495.783,Z 243.722,A -85,B 0,C 180,E1 -6153.244,E2 -6153.244} C_VEL
LIN {X 0,Y 495.684,Z 243.737,A -85,B 0,C 180,E1 -6156.084,E2 -6156.084} C_VEL
LIN {X 0,Y 495.734,Z 243.732,A -85,B 0,C 180,E1 -6158.765,E2 -6158.765} C_VEL
LIN {X 0,Y 495.718,Z 243.733,A -85,B 0,C 180,E1 -6161.785,E2 -6161.785} C_VEL
LIN {X 0,Y 495.727,Z 243.735,A -85,B 0,C 180,E1 -6165.142,E2 -6165.142} C_VEL
LIN {X 0,Y 495.718,Z 243.735,A -85,B 0,C 180,E1 -6168.216,E2 -6168.216} C_VEL
LIN {X 0,Y 495.706,Z 243.732,A -85,B 0,C 180,E1 -6171.405,E2 -6171.405} C_VEL
LIN {X 0,Y 495.724,Z 243.732,A -85,B 0,C 180,E1 -6174.461,E2 -6174.461} C_VEL
LIN {X 0,Y 495.738,Z 243.729,A -85,B 0,C 180,E1 -6177.404,E2 -6177.404} C_VEL
LIN {X 0,Y 495.693,Z 243.737,A -85,B 0,C 180,E1 -6180.249,E2 -6180.249} C_VEL
LIN {X 0,Y 495.757,Z 243.98,A -85,B 0,C 180,E1 -6181.562,E2 -6181.562} C_VEL
LIN {X 0,Y 498.291,Z 256.544,A -85,B 0,C 180,E1 -6183.397,E2 -6183.397} C_VEL
LIN {X 0,Y 497.712,Z 278.712,A -85,B 0,C 180,E1 -6186.314,E2 -6186.314} C_VEL
LIN {X 0,Y 497.041,Z 303.477,A -85,B 0,C 180,E1 -6189.515,E2 -6189.515} C_VEL
LIN {X 0,Y 496.51,Z 326.852,A -85,B 0,C 180,E1 -6192.495,E2 -6192.495} C_VEL
LIN {X 0,Y 496.266,Z 338.192,A -85,B 0,C 180,E1 -6193.912,E2 -6193.912} C_VEL
LIN {X 0,Y 498.44,Z 358.768,A -85,B 0,C 180,E1 -6194.307,E2 -6194.307} C_VEL
LIN {X 0,Y 497.9,Z 448.397,A -85,B 0,C 180,E1 -6195.621,E2 -6195.621} C_VEL
LIN {X 0,Y 497.522,Z 461.751,A -85,B 0,C 180,E1 -6195.975,E2 -6195.975} C_VEL
LIN {X 0,Y 497.152,Z 474.009,A -85,B 0,C 180,E1 -6196.459,E2 -6196.459} C_VEL
LIN {X 0,Y 496.745,Z 486.415,A -85,B 0,C 180,E1 -6197.125,E2 -6197.125} C_VEL
LIN {X 0,Y 496.416,Z 498.156,A -85,B 0,C 180,E1 -6197.947,E2 -6197.947} C_VEL
LIN {X 0,Y 495.959,Z 508.736,A -85,B 0,C 180,E1 -6198.868,E2 -6198.868} C_VEL
LIN {X 0,Y 495.704,Z 517.419,A -85,B 0,C 180,E1 -6199.792,E2 -6199.792} C_VEL
LIN {X 0,Y 495.476,Z 525.445,A -85,B 0,C 180,E1 -6200.818,E2 -6200.818} C_VEL
LIN {X 0,Y 495.326,Z 533.305,A -85,B 0,C 180,E1 -6202.048,E2 -6202.048} C_VEL
LIN {X 0,Y 495.251,Z 538.698,A -85,B 0,C 180,E1 -6203.072,E2 -6203.072} C_VEL
LIN {X 0,Y 495.22,Z 543.935,A -85,B 0,C 180,E1 -6204.299,E2 -6204.299} C_VEL
LIN {X 0,Y 495.168,Z 548.001,A -85,B 0,C 180,E1 -6205.523,E2 -6205.523} C_VEL
LIN {X 0,Y 495.196,Z 551.015,A -85,B 0,C 180,E1 -6206.745,E2 -6206.745} C_VEL
LIN {X 0,Y 495.135,Z 552.444,A -85,B 0,C 180,E1 -6207.559,E2 -6207.559} C_VEL
LIN {X 0,Y 495.102,Z 554.093,A -85,B 0,C 180,E1 -6209.186,E2 -6209.186} C_VEL
LIN {X 0,Y 495.112,Z 554.321,A -85,B 0,C 180,E1 -6210,E2 -6210} C_VEL
LIN {X 0,Y 495.101,Z 554.104,A -85,B 0,C 180,E1 -6210.813,E2 -6210.813} C_VEL
LIN {X 0,Y 495.132,Z 552.477,A -85,B 0,C 180,E1 -6212.44,E2 -6212.44} C_VEL
LIN {X 0,Y 495.194,Z 551.059,A -85,B 0,C 180,E1 -6213.254,E2 -6213.254} C_VEL
LIN {X 0,Y 495.167,Z 548.058,A -85,B 0,C 180,E1 -6214.477,E2 -6214.477} C_VEL
LIN {X 0,Y 495.207,Z 542.826,A -85,B 0,C 180,E1 -6215.998,E2 -6215.998} C_VEL
LIN {X 0,Y 495.266,Z 536.733,A -85,B 0,C 180,E1 -6217.337,E2 -6217.337} C_VEL
LIN {X 0,Y 495.388,Z 529.702,A -85,B 0,C 180,E1 -6218.566,E2 -6218.566} C_VEL
LIN {X 0,Y 495.587,Z 520.917,A -85,B 0,C 180,E1 -6219.797,E2 -6219.797} C_VEL
LIN {X 0,Y 495.913,Z 511.939,A -85,B 0,C 180,E1 -6220.822,E2 -6220.822} C_VEL
LIN {X 0,Y 496.319,Z 500.91,A -85,B 0,C 180,E1 -6221.848,E2 -6221.848} C_VEL
LIN {X 0,Y 496.676,Z 489.796,A -85,B 0,C 180,E1 -6222.668,E2 -6222.668} C_VEL
LIN {X 0,Y 497.041,Z 477.353,A -85,B 0,C 180,E1 -6223.387,E2 -6223.387} C_VEL
LIN {X 0,Y 497.415,Z 465.603,A -85,B 0,C 180,E1 -6223.897,E2 -6223.897} C_VEL
LIN {X 0,Y 497.784,Z 453.101,A -85,B 0,C 180,E1 -6224.278,E2 -6224.278} C_VEL
LIN {X 0,Y 497.97,Z 437.197,A -85,B 0,C 180,E1 -6224.559,E2 -6224.559} C_VEL
LIN {X 0,Y 498.244,Z 355.92,A -85,B 0,C 180,E1 -6225.735,E2 -6225.735} C_VEL
LIN {X 0,Y 496.263,Z 338.59,A -85,B 0,C 180,E1 -6226.063,E2 -6226.063} C_VEL
LIN {X 0,Y 496.799,Z 315.285,A -85,B 0,C 180,E1 -6228.987,E2 -6228.987} C_VEL
LIN {X 0,Y 497.426,Z 288.388,A -85,B 0,C 180,E1 -6232.424,E2 -6232.424} C_VEL
LIN {X 0,Y 497.88,Z 269.725,A -85,B 0,C 180,E1 -6234.83,E2 -6234.83} C_VEL
LIN {X 0,Y 498.201,Z 256.057,A -85,B 0,C 180,E1 -6236.607,E2 -6236.607} C_VEL
LIN {X 0,Y 495.731,Z 243.854,A -85,B 0,C 180,E1 -6238.362,E2 -6238.362} C_VEL
LIN {X 0,Y 495.726,Z 243.738,A -85,B 0,C 180,E1 -6241.719,E2 -6241.719} C_VEL
LIN {X 0,Y 495.749,Z 243.73,A -85,B 0,C 180,E1 -6244.69,E2 -6244.69} C_VEL
LIN {X 0,Y 495.686,Z 243.741,A -85,B 0,C 180,E1 -6247.564,E2 -6247.564} C_VEL
LIN {X 0,Y 495.704,Z 243.734,A -85,B 0,C 180,E1 -6250.039,E2 -6250.039} C_VEL
LIN {X 0,Y 495.681,Z 243.739,A -85,B 0,C 180,E1 -6252.886,E2 -6252.886} C_VEL
LIN {X 0,Y 495.704,Z 243.733,A -85,B 0,C 180,E1 -6255.996,E2 -6255.996} C_VEL
LIN {X 0,Y 495.716,Z 243.738,A -85,B 0,C 180,E1 -6259.295,E2 -6259.295} C_VEL
LIN {X 0,Y 495.713,Z 243.737,A -85,B 0,C 180,E1 -6261.405,E2 -6261.405} C_VEL
LIN {X 0,Y 495.718,Z 243.732,A -85,B 0,C 180,E1 -6264.46,E2 -6264.46} C_VEL
LIN {X 0,Y 495.713,Z 243.736,A -85,B 0,C 180,E1 -6267.402,E2 -6267.402} C_VEL
LIN {X 0,Y 495.726,Z 243.731,A -85,B 0,C 180,E1 -6270.251,E2 -6270.251} C_VEL
LIN {X 0,Y 495.708,Z 243.737,A -85,B 0,C 180,E1 -6273.274,E2 -6273.274} C_VEL
LIN {X 0,Y 495.691,Z 243.735,A -85,B 0,C 180,E1 -6275.722,E2 -6275.722} C_VEL
LIN {X 0,Y 495.723,Z 243.733,A -85,B 0,C 180,E1 -6278.37,E2 -6278.37} C_VEL
LIN {X 0,Y 495.75,Z 243.734,A -85,B 0,C 180,E1 -6280.97,E2 -6280.97} C_VEL
LIN {X 0,Y 495.808,Z 243.726,A -85,B 0,C 180,E1 -6284.549,E2 -6284.549} C_VEL
LIN {X 0,Y 495.815,Z 243.72,A -85,B 0,C 180,E1 -6287.965,E2 -6287.965} C_VEL
LIN {X 0,Y 495.783,Z 243.727,A -85,B 0,C 180,E1 -6291.029,E2 -6291.029} C_VEL
LIN {X 0,Y 495.789,Z 243.723,A -85,B 0,C 180,E1 -6293.489,E2 -6293.489} C_VEL
LIN {X 0,Y 495.701,Z 243.734,A -85,B 0,C 180,E1 -6295.935,E2 -6295.935} C_VEL
LIN {X 0,Y 495.964,Z 243.701,A -85,B 0,C 180,E1 -6297.564,E2 -6297.564} C_VEL
LIN {X 0,Y 495.926,Z 243.71,A -85,B 0,C 180,E1 -6300.812,E2 -6300.812} C_VEL
LIN {X 0,Y 495.958,Z 243.71,A -85,B 0,C 180,E1 -6302.437,E2 -6302.437} C_VEL
LIN {X 0,Y 495.838,Z 243.717,A -85,B 0,C 180,E1 -6305.694,E2 -6305.694} C_VEL
LIN {X 0,Y 495.795,Z 243.727,A -85,B 0,C 180,E1 -6308.149,E2 -6308.149} C_VEL
LIN {X 0,Y 495.806,Z 243.72,A -85,B 0,C 180,E1 -6311.446,E2 -6311.446} C_VEL
LIN {X 0,Y 495.769,Z 243.727,A -85,B 0,C 180,E1 -6314.784,E2 -6314.784} C_VEL
LIN {X 0,Y 495.767,Z 243.734,A -85,B 0,C 180,E1 -6318.172,E2 -6318.172} C_VEL
LIN {X 0,Y 495.762,Z 243.727,A -85,B 0,C 180,E1 -6320.757,E2 -6320.757} C_VEL
LIN {X 0,Y 495.727,Z 243.731,A -85,B 0,C 180,E1 -6323.389,E2 -6323.389} C_VEL
LIN {X 0,Y 495.726,Z 243.731,A -85,B 0,C 180,E1 -6326.73,E2 -6326.73} C_VEL
LIN {X 0,Y 495.745,Z 243.733,A -85,B 0,C 180,E1 -6329.748,E2 -6329.748} C_VEL
LIN {X 0,Y 495.733,Z 243.731,A -85,B 0,C 180,E1 -6332.597,E2 -6332.597} C_VEL
LIN {X 0,Y 495.718,Z 243.735,A -85,B 0,C 180,E1 -6335.541,E2 -6335.541} C_VEL
LIN {X 0,Y 495.72,Z 243.731,A -85,B 0,C 180,E1 -6338.764,E2 -6338.764} C_VEL
LIN {X 0,Y 495.692,Z 243.743,A -85,B 0,C 180,E1 -6341.788,E2 -6341.788} C_VEL
LIN {X 0,Y 495.725,Z 243.732,A -85,B 0,C 180,E1 -6345.143,E2 -6345.143} C_VEL
LIN {X 0,Y 495.697,Z 243.736,A -85,B 0,C 180,E1 -6348.214,E2 -6348.214} C_VEL
LIN {X 0,Y 495.711,Z 243.737,A -85,B 0,C 180,E1 -6351.406,E2 -6351.406} C_VEL
LIN {X 0,Y 495.712,Z 243.732,A -85,B 0,C 180,E1 -6354.461,E2 -6354.461} C_VEL
LIN {X 0,Y 495.722,Z 243.737,A -85,B 0,C 180,E1 -6357.404,E2 -6357.404} C_VEL
LIN {X 0,Y 495.697,Z 243.734,A -85,B 0,C 180,E1 -6360.25,E2 -6360.25} C_VEL
LIN {X 0,Y 495.681,Z 243.736,A -85,B 0,C 180,E1 -6360.761,E2 -6360.761} C_VEL
LIN {X 0,Y 495.02,Z 243.826,A -85,B 0,C 180,E1 -6361.44,E2 -6361.44} C_VEL
LIN {X 0,Y 492.156,Z 244.179,A -85,B 0,C 180,E1 -6362.542,E2 -6362.542} C_VEL
LIN {X 0,Y 489.741,Z 244.484,A -85,B 0,C 180,E1 -6363.431,E2 -6363.431} C_VEL
LIN {X 0,Y 488.72,Z 244.605,A -85,B 0,C 180,E1 -6364.117,E2 -6364.117} C_VEL
LIN {X 0,Y 488.646,Z 244.612,A -85,B 0,C 180,E1 -6364.349,E2 -6364.349} C_VEL
LIN {X 0,Y 488.708,Z 244.61,A -85,B 0,C 180,E1 -6367.153,E2 -6367.153} C_VEL
LIN {X 0,Y 488.695,Z 244.609,A -85,B 0,C 180,E1 -6369.81,E2 -6369.81} C_VEL
LIN {X 0,Y 488.69,Z 244.607,A -85,B 0,C 180,E1 -6372.423,E2 -6372.423} C_VEL
LIN {X 0,Y 488.716,Z 244.608,A -85,B 0,C 180,E1 -6374.999,E2 -6374.999} C_VEL
LIN {X 0,Y 488.788,Z 244.597,A -85,B 0,C 180,E1 -6378.388,E2 -6378.388} C_VEL
LIN {X 0,Y 488.805,Z 244.741,A -85,B 0,C 180,E1 -6381.941,E2 -6381.941} C_VEL
LIN {X 0,Y 488.966,Z 245.605,A -85,B 0,C 180,E1 -6382.078,E2 -6382.078} C_VEL
LIN {X 0,Y 491.8,Z 253.614,A -85,B 0,C 180,E1 -6382.308,E2 -6382.308} C_VEL
LIN {X 0,Y 491.339,Z 333.733,A -85,B 0,C 180,E1 -6383.507,E2 -6383.507} C_VEL
LIN {X 0,Y 491.203,Z 347.303,A -85,B 0,C 180,E1 -6383.892,E2 -6383.892} C_VEL
LIN {X 0,Y 491.034,Z 359.5,A -85,B 0,C 180,E1 -6384.405,E2 -6384.405} C_VEL
LIN {X 0,Y 490.725,Z 371.216,A -85,B 0,C 180,E1 -6385.071,E2 -6385.071} C_VEL
LIN {X 0,Y 490.345,Z 382.439,A -85,B 0,C 180,E1 -6385.891,E2 -6385.891} C_VEL
LIN {X 0,Y 489.955,Z 392.56,A -85,B 0,C 180,E1 -6386.814,E2 -6386.814} C_VEL
LIN {X 0,Y 489.662,Z 400.835,A -85,B 0,C 180,E1 -6387.738,E2 -6387.738} C_VEL
LIN {X 0,Y 489.31,Z 409.822,A -85,B 0,C 180,E1 -6388.972,E2 -6388.972} C_VEL
LIN {X 0,Y 488.929,Z 417.072,A -85,B 0,C 180,E1 -6390.206,E2 -6390.206} C_VEL
LIN {X 0,Y 488.633,Z 423.756,A -85,B 0,C 180,E1 -6391.649,E2 -6391.649} C_VEL
LIN {X 0,Y 488.484,Z 428.162,A -85,B 0,C 180,E1 -6392.887,E2 -6392.887} C_VEL
LIN {X 0,Y 488.399,Z 431.518,A -85,B 0,C 180,E1 -6394.126,E2 -6394.126} C_VEL
LIN {X 0,Y 488.428,Z 433.179,A -85,B 0,C 180,E1 -6394.953,E2 -6394.953} C_VEL
LIN {X 0,Y 488.341,Z 435.36,A -85,B 0,C 180,E1 -6396.611,E2 -6396.611} C_VEL
LIN {X 0,Y 488.31,Z 435.859,A -85,B 0,C 180,E1 -6397.443,E2 -6397.443} C_VEL
LIN {X 0,Y 488.285,Z 435.646,A -85,B 0,C 180,E1 -6399.11,E2 -6399.11} C_VEL
LIN {X 0,Y 488.289,Z 434.969,A -85,B 0,C 180,E1 -6399.946,E2 -6399.946} C_VEL
LIN {X 0,Y 488.343,Z 433.868,A -85,B 0,C 180,E1 -6400.783,E2 -6400.783} C_VEL
LIN {X 0,Y 488.462,Z 431.68,A -85,B 0,C 180,E1 -6401.932,E2 -6401.932} C_VEL
LIN {X 0,Y 488.568,Z 427.976,A -85,B 0,C 180,E1 -6403.306,E2 -6403.306} C_VEL
LIN {X 0,Y 488.746,Z 423.385,A -85,B 0,C 180,E1 -6404.575,E2 -6404.575} C_VEL
LIN {X 0,Y 489.034,Z 416.387,A -85,B 0,C 180,E1 -6406.06,E2 -6406.06} C_VEL
LIN {X 0,Y 489.407,Z 408.729,A -85,B 0,C 180,E1 -6407.336,E2 -6407.336} C_VEL
LIN {X 0,Y 489.724,Z 400.798,A -85,B 0,C 180,E1 -6408.404,E2 -6408.404} C_VEL
LIN {X 0,Y 490.131,Z 391.041,A -85,B 0,C 180,E1 -6409.474,E2 -6409.474} C_VEL
LIN {X 0,Y 490.501,Z 380.095,A -85,B 0,C 180,E1 -6410.441,E2 -6410.441} C_VEL
LIN {X 0,Y 490.913,Z 368.885,A -85,B 0,C 180,E1 -6411.215,E2 -6411.215} C_VEL
LIN {X 0,Y 491.195,Z 356.1,A -85,B 0,C 180,E1 -6411.894,E2 -6411.894} C_VEL
LIN {X 0,Y 491.354,Z 343.225,A -85,B 0,C 180,E1 -6412.385,E2 -6412.385} C_VEL
LIN {X 0,Y 491.519,Z 329.429,A -85,B 0,C 180,E1 -6412.709,E2 -6412.709} C_VEL
LIN {X 0,Y 491.978,Z 254.074,A -85,B 0,C 180,E1 -6413.83,E2 -6413.83} C_VEL
LIN {X 0,Y 488.844,Z 245.428,A -85,B 0,C 180,E1 -6414.108,E2 -6414.108} C_VEL
LIN {X 0,Y 488.694,Z 244.665,A -85,B 0,C 180,E1 -6414.293,E2 -6414.293} C_VEL
LIN {X 0,Y 488.688,Z 244.612,A -85,B 0,C 180,E1 -6417.4,E2 -6417.4} C_VEL
LIN {X 0,Y 488.709,Z 244.6,A -85,B 0,C 180,E1 -6420.362,E2 -6420.362} C_VEL
LIN {X 0,Y 488.711,Z 244.608,A -85,B 0,C 180,E1 -6423.479,E2 -6423.479} C_VEL
LIN {X 0,Y 488.668,Z 244.595,A -85,B 0,C 180,E1 -6426.351,E2 -6426.351} C_VEL
LIN {X 0,Y 488.687,Z 244.611,A -85,B 0,C 180,E1 -6429.255,E2 -6429.255} C_VEL
LIN {X 0,Y 488.666,Z 244.612,A -85,B 0,C 180,E1 -6432.528,E2 -6432.528} C_VEL
LIN {X 0,Y 488.7,Z 244.607,A -85,B 0,C 180,E1 -6435.197,E2 -6435.197} C_VEL
LIN {X 0,Y 488.66,Z 244.617,A -85,B 0,C 180,E1 -6438.579,E2 -6438.579} C_VEL
LIN {X 0,Y 488.685,Z 244.606,A -85,B 0,C 180,E1 -6440.949,E2 -6440.949} C_VEL
LIN {X 0,Y 488.649,Z 244.609,A -85,B 0,C 180,E1 -6443.865,E2 -6443.865} C_VEL
LIN {X 0,Y 488.733,Z 244.603,A -85,B 0,C 180,E1 -6446.876,E2 -6446.876} C_VEL
LIN {X 0,Y 488.718,Z 244.594,A -85,B 0,C 180,E1 -6449.78,E2 -6449.78} C_VEL
LIN {X 0,Y 488.693,Z 244.608,A -85,B 0,C 180,E1 -6453.078,E2 -6453.078} C_VEL
LIN {X 0,Y 488.667,Z 244.606,A -85,B 0,C 180,E1 -6456.253,E2 -6456.253} C_VEL
LIN {X 0,Y 488.741,Z 244.588,A -85,B 0,C 180,E1 -6459.175,E2 -6459.175} C_VEL
LIN {X 0,Y 488.741,Z 244.601,A -85,B 0,C 180,E1 -6461.632,E2 -6461.632} C_VEL
LIN {X 0,Y 488.749,Z 244.596,A -85,B 0,C 180,E1 -6464.999,E2 -6464.999} C_VEL
LIN {X 0,Y 488.797,Z 244.596,A -85,B 0,C 180,E1 -6468.387,E2 -6468.387} C_VEL
LIN {X 0,Y 488.753,Z 244.601,A -85,B 0,C 180,E1 -6471.732,E2 -6471.732} C_VEL
LIN {X 0,Y 488.806,Z 244.594,A -85,B 0,C 180,E1 -6474.223,E2 -6474.223} C_VEL
LIN {X 0,Y 488.932,Z 244.579,A -85,B 0,C 180,E1 -6477.528,E2 -6477.528} C_VEL
LIN {X 0,Y 488.93,Z 244.579,A -85,B 0,C 180,E1 -6480,E2 -6480} C_VEL
LIN {X 0,Y 488.939,Z 244.573,A -85,B 0,C 180,E1 -6482.471,E2 -6482.471} C_VEL
LIN {X 0,Y 488.796,Z 244.597,A -85,B 0,C 180,E1 -6485.776,E2 -6485.776} C_VEL
LIN {X 0,Y 488.769,Z 244.595,A -85,B 0,C 180,E1 -6488.267,E2 -6488.267} C_VEL
LIN {X 0,Y 488.795,Z 244.597,A -85,B 0,C 180,E1 -6491.613,E2 -6491.613} C_VEL
LIN {X 0,Y 488.744,Z 244.603,A -85,B 0,C 180,E1 -6495.001,E2 -6495.001} C_VEL
LIN {X 0,Y 488.737,Z 244.599,A -85,B 0,C 180,E1 -6498.443,E2 -6498.443} C_VEL
LIN {X 0,Y 488.699,Z 244.613,A -85,B 0,C 180,E1 -6501.071,E2 -6501.071} C_VEL
LIN {X 0,Y 488.66,Z 244.614,A -85,B 0,C 180,E1 -6503.747,E2 -6503.747} C_VEL
LIN {X 0,Y 488.689,Z 244.606,A -85,B 0,C 180,E1 -6506.922,E2 -6506.922} C_VEL
LIN {X 0,Y 488.691,Z 244.608,A -85,B 0,C 180,E1 -6510.222,E2 -6510.222} C_VEL
LIN {X 0,Y 488.706,Z 244.601,A -85,B 0,C 180,E1 -6513.48,E2 -6513.48} C_VEL
LIN {X 0,Y 488.646,Z 244.615,A -85,B 0,C 180,E1 -6516.35,E2 -6516.35} C_VEL
LIN {X 0,Y 488.682,Z 244.612,A -85,B 0,C 180,E1 -6519.256,E2 -6519.256} C_VEL
LIN {X 0,Y 488.662,Z 244.613,A -85,B 0,C 180,E1 -6521.595,E2 -6521.595} C_VEL
LIN {X 0,Y 488.691,Z 244.615,A -85,B 0,C 180,E1 -6524.804,E2 -6524.804} C_VEL
LIN {X 0,Y 488.644,Z 244.615,A -85,B 0,C 180,E1 -6527.47,E2 -6527.47} C_VEL
LIN {X 0,Y 488.665,Z 244.605,A -85,B 0,C 180,E1 -6530.743,E2 -6530.743} C_VEL
LIN {X 0,Y 488.639,Z 244.616,A -85,B 0,C 180,E1 -6533.865,E2 -6533.865} C_VEL
LIN {X 0,Y 488.706,Z 244.613,A -85,B 0,C 180,E1 -6536.521,E2 -6536.521} C_VEL
LIN {X 0,Y 488.661,Z 244.616,A -85,B 0,C 180,E1 -6539.777,E2 -6539.777} C_VEL
LIN {X 0,Y 488.692,Z 244.779,A -85,B 0,C 180,E1 -6541.313,E2 -6541.313} C_VEL
LIN {X 0,Y 491.333,Z 257.515,A -85,B 0,C 180,E1 -6543.22,E2 -6543.22} C_VEL
LIN {X 0,Y 491.073,Z 269.271,A -85,B 0,C 180,E1 -6544.801,E2 -6544.801} C_VEL
LIN {X 0,Y 490.457,Z 289.357,A -85,B 0,C 180,E1 -6547.461,E2 -6547.461} C_VEL
LIN {X 0,Y 489.821,Z 312.709,A -85,B 0,C 180,E1 -6550.513,E2 -6550.513} C_VEL
LIN {X 0,Y 489.248,Z 335.866,A -85,B 0,C 180,E1 -6553.497,E2 -6553.497} C_VEL
LIN {X 0,Y 489.235,Z 337.402,A -85,B 0,C 180,E1 -6553.672,E2 -6553.672} C_VEL
LIN {X 0,Y 491.587,Z 359.151,A -85,B 0,C 180,E1 -6554.094,E2 -6554.094} C_VEL
LIN {X 0,Y 490.995,Z 447.792,A -85,B 0,C 180,E1 -6555.414,E2 -6555.414} C_VEL
LIN {X 0,Y 490.664,Z 461.04,A -85,B 0,C 180,E1 -6555.775,E2 -6555.775} C_VEL
LIN {X 0,Y 490.224,Z 473.239,A -85,B 0,C 180,E1 -6556.264,E2 -6556.264} C_VEL
LIN {X 0,Y 489.785,Z 485.601,A -85,B 0,C 180,E1 -6556.939,E2 -6556.939} C_VEL
LIN {X 0,Y 489.42,Z 496.456,A -85,B 0,C 180,E1 -6557.703,E2 -6557.703} C_VEL
LIN {X 0,Y 488.968,Z 507.88,A -85,B 0,C 180,E1 -6558.706,E2 -6558.706} C_VEL
LIN {X 0,Y 488.662,Z 516.554,A -85,B 0,C 180,E1 -6559.643,E2 -6559.643} C_VEL
LIN {X 0,Y 488.418,Z 524.576,A -85,B 0,C 180,E1 -6560.684,E2 -6560.684} C_VEL
LIN {X 0,Y 488.246,Z 532.435,A -85,B 0,C 180,E1 -6561.932,E2 -6561.932} C_VEL
LIN {X 0,Y 488.18,Z 537.831,A -85,B 0,C 180,E1 -6562.971,E2 -6562.971} C_VEL
LIN {X 0,Y 488.155,Z 543.073,A -85,B 0,C 180,E1 -6564.216,E2 -6564.216} C_VEL
LIN {X 0,Y 488.104,Z 547.143,A -85,B 0,C 180,E1 -6565.458,E2 -6565.458} C_VEL
LIN {X 0,Y 488.143,Z 550.161,A -85,B 0,C 180,E1 -6566.698,E2 -6566.698} C_VEL
LIN {X 0,Y 488.079,Z 551.591,A -85,B 0,C 180,E1 -6567.524,E2 -6567.524} C_VEL
LIN {X 0,Y 488.051,Z 553.244,A -85,B 0,C 180,E1 -6569.175,E2 -6569.175} C_VEL
LIN {X 0,Y 488.063,Z 553.473,A -85,B 0,C 180,E1 -6570,E2 -6570} C_VEL
LIN {X 0,Y 488.05,Z 553.256,A -85,B 0,C 180,E1 -6570.825,E2 -6570.825} C_VEL
LIN {X 0,Y 488.076,Z 551.63,A -85,B 0,C 180,E1 -6572.475,E2 -6572.475} C_VEL
LIN {X 0,Y 488.141,Z 550.212,A -85,B 0,C 180,E1 -6573.301,E2 -6573.301} C_VEL
LIN {X 0,Y 488.103,Z 547.209,A -85,B 0,C 180,E1 -6574.542,E2 -6574.542} C_VEL
LIN {X 0,Y 488.153,Z 543.155,A -85,B 0,C 180,E1 -6575.784,E2 -6575.784} C_VEL
LIN {X 0,Y 488.178,Z 536.912,A -85,B 0,C 180,E1 -6577.236,E2 -6577.236} C_VEL
LIN {X 0,Y 488.293,Z 530.107,A -85,B 0,C 180,E1 -6578.483,E2 -6578.483} C_VEL
LIN {X 0,Y 488.474,Z 521.673,A -85,B 0,C 180,E1 -6579.732,E2 -6579.732} C_VEL
LIN {X 0,Y 488.802,Z 513.051,A -85,B 0,C 180,E1 -6580.772,E2 -6580.772} C_VEL
LIN {X 0,Y 489.203,Z 502.541,A -85,B 0,C 180,E1 -6581.801,E2 -6581.801} C_VEL
LIN {X 0,Y 489.627,Z 490.611,A -85,B 0,C 180,E1 -6582.738,E2 -6582.738} C_VEL
LIN {X 0,Y 490.04,Z 478.433,A -85,B 0,C 180,E1 -6583.476,E2 -6583.476} C_VEL
LIN {X 0,Y 490.444,Z 465.945,A -85,B 0,C 180,E1 -6584.046,E2 -6584.046} C_VEL
LIN {X 0,Y 490.856,Z 453.115,A -85,B 0,C 180,E1 -6584.457,E2 -6584.457} C_VEL
LIN {X 0,Y 491.077,Z 439.556,A -85,B 0,C 180,E1 -6584.715,E2 -6584.715} C_VEL
LIN {X 0,Y 491.382,Z 356.709,A -85,B 0,C 180,E1 -6585.925,E2 -6585.925} C_VEL
LIN {X 0,Y 489.244,Z 337.687,A -85,B 0,C 180,E1 -6586.295,E2 -6586.295} C_VEL
LIN {X 0,Y 489.797,Z 314.328,A -85,B 0,C 180,E1 -6589.269,E2 -6589.269} C_VEL
LIN {X 0,Y 490.438,Z 289.082,A -85,B 0,C 180,E1 -6592.539,E2 -6592.539} C_VEL
LIN {X 0,Y 490.939,Z 270.405,A -85,B 0,C 180,E1 -6594.979,E2 -6594.979} C_VEL
LIN {X 0,Y 491.289,Z 258.454,A -85,B 0,C 180,E1 -6596.553,E2 -6596.553} C_VEL
LIN {X 0,Y 490.082,Z 251.39,A -85,B 0,C 180,E1 -6597.546,E2 -6597.546} C_VEL
LIN {X 0,Y 488.678,Z 244.732,A -85,B 0,C 180,E1 -6598.539,E2 -6598.539} C_VEL
LIN {X 0,Y 488.653,Z 244.616,A -85,B 0,C 180,E1 -6601.181,E2 -6601.181} C_VEL
LIN {X 0,Y 488.71,Z 244.608,A -85,B 0,C 180,E1 -6604.113,E2 -6604.113} C_VEL
LIN {X 0,Y 488.636,Z 244.619,A -85,B 0,C 180,E1 -6607.161,E2 -6607.161} C_VEL
LIN {X 0,Y 488.66,Z 244.61,A -85,B 0,C 180,E1 -6610.329,E2 -6610.329} C_VEL
LIN {X 0,Y 488.656,Z 244.614,A -85,B 0,C 180,E1 -6613.656,E2 -6613.656} C_VEL
LIN {X 0,Y 488.656,Z 244.611,A -85,B 0,C 180,E1 -6616.342,E2 -6616.342} C_VEL
LIN {X 0,Y 488.694,Z 244.608,A -85,B 0,C 180,E1 -6619.673,E2 -6619.673} C_VEL
LIN {X 0,Y 488.64,Z 244.618,A -85,B 0,C 180,E1 -6622.838,E2 -6622.838} C_VEL
LIN {X 0,Y 488.698,Z 244.606,A -85,B 0,C 180,E1 -6625.885,E2 -6625.885} C_VEL
LIN {X 0,Y 488.654,Z 244.617,A -85,B 0,C 180,E1 -6628.818,E2 -6628.818} C_VEL
LIN {X 0,Y 488.679,Z 244.609,A -85,B 0,C 180,E1 -6631.667,E2 -6631.667} C_VEL
LIN {X 0,Y 488.68,Z 244.616,A -85,B 0,C 180,E1 -6634.96,E2 -6634.96} C_VEL
LIN {X 0,Y 488.68,Z 244.608,A -85,B 0,C 180,E1 -6638.042,E2 -6638.042} C_VEL
LIN {X 0,Y 488.713,Z 244.61,A -85,B 0,C 180,E1 -6640.686,E2 -6640.686} C_VEL
LIN {X 0,Y 488.74,Z 244.602,A -85,B 0,C 180,E1 -6644.144,E2 -6644.144} C_VEL
LIN {X 0,Y 488.721,Z 244.603,A -85,B 0,C 180,E1 -6647.543,E2 -6647.543} C_VEL
LIN {X 0,Y 488.726,Z 244.604,A -85,B 0,C 180,E1 -6650.063,E2 -6650.063} C_VEL
LIN {X 0,Y 488.803,Z 244.599,A -85,B 0,C 180,E1 -6652.771,E2 -6652.771} C_VEL
LIN {X 0,Y 488.767,Z 244.6,A -85,B 0,C 180,E1 -6655.051,E2 -6655.051} C_VEL
LIN {X 0,Y 488.932,Z 244.577,A -85,B 0,C 180,E1 -6657.529,E2 -6657.529} C_VEL
LIN {X 0,Y 488.878,Z 244.587,A -85,B 0,C 180,E1 -6660.824,E2 -6660.824} C_VEL
LIN {X 0,Y 488.924,Z 244.586,A -85,B 0,C 180,E1 -6662.472,E2 -6662.472} C_VEL
LIN {X 0,Y 488.798,Z 244.595,A -85,B 0,C 180,E1 -6665.777,E2 -6665.777} C_VEL
LIN {X 0,Y 488.74,Z 244.608,A -85,B 0,C 180,E1 -6668.268,E2 -6668.268} C_VEL
LIN {X 0,Y 488.769,Z 244.598,A -85,B 0,C 180,E1 -6671.614,E2 -6671.614} C_VEL
LIN {X 0,Y 488.744,Z 244.601,A -85,B 0,C 180,E1 -6675.001,E2 -6675.001} C_VEL
LIN {X 0,Y 488.732,Z 244.607,A -85,B 0,C 180,E1 -6678.443,E2 -6678.443} C_VEL
LIN {X 0,Y 488.694,Z 244.606,A -85,B 0,C 180,E1 -6681.072,E2 -6681.072} C_VEL
LIN {X 0,Y 488.658,Z 244.614,A -85,B 0,C 180,E1 -6683.748,E2 -6683.748} C_VEL
LIN {X 0,Y 488.684,Z 244.608,A -85,B 0,C 180,E1 -6686.922,E2 -6686.922} C_VEL
LIN {X 0,Y 488.706,Z 244.61,A -85,B 0,C 180,E1 -6690.221,E2 -6690.221} C_VEL
LIN {X 0,Y 488.698,Z 244.608,A -85,B 0,C 180,E1 -6693.48,E2 -6693.48} C_VEL
LIN {X 0,Y 488.639,Z 244.616,A -85,B 0,C 180,E1 -6696.35,E2 -6696.35} C_VEL
LIN {X 0,Y 488.66,Z 244.612,A -85,B 0,C 180,E1 -6699.259,E2 -6699.259} C_VEL
LIN {X 0,Y 488.64,Z 244.614,A -85,B 0,C 180,E1 -6702.532,E2 -6702.532} C_VEL
LIN {X 0,Y 488.69,Z 244.608,A -85,B 0,C 180,E1 -6705.198,E2 -6705.198} C_VEL
LIN {X 0,Y 488.639,Z 244.613,A -85,B 0,C 180,E1 -6708.579,E2 -6708.579} C_VEL
LIN {X 0,Y 488.646,Z 244.619,A -85,B 0,C 180,E1 -6711.798,E2 -6711.798} C_VEL
LIN {X 0,Y 488.699,Z 244.608,A -85,B 0,C 180,E1 -6715.058,E2 -6715.058} C_VEL
LIN {X 0,Y 488.681,Z 244.61,A -85,B 0,C 180,E1 -6718.051,E2 -6718.051} C_VEL
LIN {X 0,Y 488.662,Z 244.616,A -85,B 0,C 180,E1 -6721.321,E2 -6721.321} C_VEL
LIN {X 0,Y 488.646,Z 244.612,A -85,B 0,C 180,E1 -6724.349,E2 -6724.349} C_VEL
LIN {X 0,Y 488.006,Z 244.697,A -85,B 0,C 180,E1 -6725.037,E2 -6725.037} C_VEL
LIN {X 0,Y 485.17,Z 245.049,A -85,B 0,C 180,E1 -6726.155,E2 -6726.155} C_VEL
LIN {X 0,Y 482.753,Z 245.351,A -85,B 0,C 180,E1 -6727.056,E2 -6727.056} C_VEL
LIN {X 0,Y 481.711,Z 245.48,A -85,B 0,C 180,E1 -6727.752,E2 -6727.752} C_VEL
LIN {X 0,Y 481.624,Z 245.488,A -85,B 0,C 180,E1 -6727.988,E2 -6727.988} C_VEL
LIN {X 0,Y 481.657,Z 245.483,A -85,B 0,C 180,E1 -6730.392,E2 -6730.392} C_VEL
LIN {X 0,Y 481.656,Z 245.488,A -85,B 0,C 180,E1 -6733.033,E2 -6733.033} C_VEL
LIN {X 0,Y 481.647,Z 245.487,A -85,B 0,C 180,E1 -6735.638,E2 -6735.638} C_VEL
LIN {X 0,Y 481.739,Z 245.475,A -85,B 0,C 180,E1 -6738.215,E2 -6738.215} C_VEL
LIN {X 0,Y 481.727,Z 245.6,A -85,B 0,C 180,E1 -6741.709,E2 -6741.709} C_VEL
LIN {X 0,Y 481.951,Z 246.542,A -85,B 0,C 180,E1 -6741.863,E2 -6741.863} C_VEL
LIN {X 0,Y 485,Z 255.683,A -85,B 0,C 180,E1 -6742.118,E2 -6742.118} C_VEL
LIN {X 0,Y 484.467,Z 334.486,A -85,B 0,C 180,E1 -6743.31,E2 -6743.31} C_VEL
LIN {X 0,Y 484.347,Z 348.075,A -85,B 0,C 180,E1 -6743.701,E2 -6743.701} C_VEL
LIN {X 0,Y 484.161,Z 360.296,A -85,B 0,C 180,E1 -6744.221,E2 -6744.221} C_VEL
LIN {X 0,Y 483.853,Z 372.022,A -85,B 0,C 180,E1 -6744.896,E2 -6744.896} C_VEL
LIN {X 0,Y 483.445,Z 383.259,A -85,B 0,C 180,E1 -6745.728,E2 -6745.728} C_VEL
LIN {X 0,Y 483.048,Z 393.387,A -85,B 0,C 180,E1 -6746.664,E2 -6746.664} C_VEL
LIN {X 0,Y 482.672,Z 402.507,A -85,B 0,C 180,E1 -6747.706,E2 -6747.706} C_VEL
LIN {X 0,Y 482.321,Z 411.322,A -85,B 0,C 180,E1 -6748.957,E2 -6748.957} C_VEL
LIN {X 0,Y 481.912,Z 418.463,A -85,B 0,C 180,E1 -6750.209,E2 -6750.209} C_VEL
LIN {X 0,Y 481.613,Z 424.996,A -85,B 0,C 180,E1 -6751.673,E2 -6751.673} C_VEL
LIN {X 0,Y 481.456,Z 429.313,A -85,B 0,C 180,E1 -6752.929,E2 -6752.929} C_VEL
LIN {X 0,Y 481.361,Z 432.587,A -85,B 0,C 180,E1 -6754.187,E2 -6754.187} C_VEL
LIN {X 0,Y 481.374,Z 434.208,A -85,B 0,C 180,E1 -6755.026,E2 -6755.026} C_VEL
LIN {X 0,Y 481.312,Z 436.301,A -85,B 0,C 180,E1 -6756.708,E2 -6756.708} C_VEL
LIN {X 0,Y 481.229,Z 436.774,A -85,B 0,C 180,E1 -6758.398,E2 -6758.398} C_VEL
LIN {X 0,Y 481.259,Z 436.435,A -85,B 0,C 180,E1 -6759.244,E2 -6759.244} C_VEL
LIN {X 0,Y 481.252,Z 435.712,A -85,B 0,C 180,E1 -6760.093,E2 -6760.093} C_VEL
LIN {X 0,Y 481.338,Z 434.536,A -85,B 0,C 180,E1 -6760.942,E2 -6760.942} C_VEL
LIN {X 0,Y 481.436,Z 432.49,A -85,B 0,C 180,E1 -6762.02,E2 -6762.02} C_VEL
LIN {X 0,Y 481.566,Z 428.473,A -85,B 0,C 180,E1 -6763.504,E2 -6763.504} C_VEL
LIN {X 0,Y 481.786,Z 423.784,A -85,B 0,C 180,E1 -6764.79,E2 -6764.79} C_VEL
LIN {X 0,Y 482.052,Z 417.798,A -85,B 0,C 180,E1 -6766.082,E2 -6766.082} C_VEL
LIN {X 0,Y 482.43,Z 410.284,A -85,B 0,C 180,E1 -6767.376,E2 -6767.376} C_VEL
LIN {X 0,Y 482.79,Z 402.545,A -85,B 0,C 180,E1 -6768.458,E2 -6768.458} C_VEL
LIN {X 0,Y 483.203,Z 392.998,A -85,B 0,C 180,E1 -6769.544,E2 -6769.544} C_VEL
LIN {X 0,Y 483.582,Z 382.297,A -85,B 0,C 180,E1 -6770.525,E2 -6770.525} C_VEL
LIN {X 0,Y 484.01,Z 371.892,A -85,B 0,C 180,E1 -6771.285,E2 -6771.285} C_VEL
LIN {X 0,Y 484.35,Z 360.948,A -85,B 0,C 180,E1 -6771.917,E2 -6771.917} C_VEL
LIN {X 0,Y 484.542,Z 348.243,A -85,B 0,C 180,E1 -6772.464,E2 -6772.464} C_VEL
LIN {X 0,Y 484.667,Z 334.799,A -85,B 0,C 180,E1 -6772.851,E2 -6772.851} C_VEL
LIN {X 0,Y 484.938,Z 297.53,A -85,B 0,C 180,E1 -6773.432,E2 -6773.432} C_VEL
LIN {X 0,Y 485.187,Z 255.361,A -85,B 0,C 180,E1 -6774.067,E2 -6774.067} C_VEL
LIN {X 0,Y 481.849,Z 246.405,A -85,B 0,C 180,E1 -6774.363,E2 -6774.363} C_VEL
LIN {X 0,Y 481.669,Z 245.547,A -85,B 0,C 180,E1 -6774.544,E2 -6774.544} C_VEL
LIN {X 0,Y 481.655,Z 245.487,A -85,B 0,C 180,E1 -6777.834,E2 -6777.834} C_VEL
LIN {X 0,Y 481.645,Z 245.476,A -85,B 0,C 180,E1 -6780.711,E2 -6780.711} C_VEL
LIN {X 0,Y 481.677,Z 245.484,A -85,B 0,C 180,E1 -6783.728,E2 -6783.728} C_VEL
LIN {X 0,Y 481.616,Z 245.473,A -85,B 0,C 180,E1 -6786.747,E2 -6786.747} C_VEL
LIN {X 0,Y 481.655,Z 245.487,A -85,B 0,C 180,E1 -6789.942,E2 -6789.942} C_VEL
LIN {X 0,Y 481.621,Z 245.49,A -85,B 0,C 180,E1 -6793.301,E2 -6793.301} C_VEL
LIN {X 0,Y 481.65,Z 245.484,A -85,B 0,C 180,E1 -6795.641,E2 -6795.641} C_VEL
LIN {X 0,Y 481.621,Z 245.491,A -85,B 0,C 180,E1 -6798.954,E2 -6798.954} C_VEL
LIN {X 0,Y 481.628,Z 245.484,A -85,B 0,C 180,E1 -6801.996,E2 -6801.996} C_VEL
LIN {X 0,Y 481.68,Z 245.482,A -85,B 0,C 180,E1 -6805.317,E2 -6805.317} C_VEL
LIN {X 0,Y 481.64,Z 245.481,A -85,B 0,C 180,E1 -6808.311,E2 -6808.311} C_VEL
LIN {X 0,Y 481.659,Z 245.478,A -85,B 0,C 180,E1 -6811.215,E2 -6811.215} C_VEL
LIN {X 0,Y 481.641,Z 245.493,A -85,B 0,C 180,E1 -6814.039,E2 -6814.039} C_VEL
LIN {X 0,Y 481.669,Z 245.471,A -85,B 0,C 180,E1 -6816.811,E2 -6816.811} C_VEL
LIN {X 0,Y 481.689,Z 245.467,A -85,B 0,C 180,E1 -6819.502,E2 -6819.502} C_VEL
LIN {X 0,Y 481.68,Z 245.487,A -85,B 0,C 180,E1 -6822.157,E2 -6822.157} C_VEL
LIN {X 0,Y 481.732,Z 245.471,A -85,B 0,C 180,E1 -6824.775,E2 -6824.775} C_VEL
LIN {X 0,Y 481.743,Z 245.476,A -85,B 0,C 180,E1 -6828.215,E2 -6828.215} C_VEL
LIN {X 0,Y 481.712,Z 245.476,A -85,B 0,C 180,E1 -6831.611,E2 -6831.611} C_VEL
LIN {X 0,Y 481.767,Z 245.472,A -85,B 0,C 180,E1 -6834.139,E2 -6834.139} C_VEL
LIN {X 0,Y 481.898,Z 245.454,A -85,B 0,C 180,E1 -6837.492,E2 -6837.492} C_VEL
LIN {X 0,Y 481.9,Z 245.455,A -85,B 0,C 180,E1 -6840,E2 -6840} C_VEL
LIN {X 0,Y 481.906,Z 245.449,A -85,B 0,C 180,E1 -6842.507,E2 -6842.507} C_VEL
LIN {X 0,Y 481.757,Z 245.472,A -85,B 0,C 180,E1 -6845.861,E2 -6845.861} C_VEL
LIN {X 0,Y 481.725,Z 245.472,A -85,B 0,C 180,E1 -6848.389,E2 -6848.389} C_VEL
LIN {X 0,Y 481.742,Z 245.473,A -85,B 0,C 180,E1 -6851.785,E2 -6851.785} C_VEL
LIN {X 0,Y 481.728,Z 245.479,A -85,B 0,C 180,E1 -6855.225,E2 -6855.225} C_VEL
LIN {X 0,Y 481.698,Z 245.477,A -85,B 0,C 180,E1 -6858.722,E2 -6858.722} C_VEL
LIN {X 0,Y 481.637,Z 245.49,A -85,B 0,C 180,E1 -6861.395,E2 -6861.395} C_VEL
LIN {X 0,Y 481.64,Z 245.487,A -85,B 0,C 180,E1 -6864.115,E2 -6864.115} C_VEL
LIN {X 0,Y 481.644,Z 245.481,A -85,B 0,C 180,E1 -6867.117,E2 -6867.117} C_VEL
LIN {X 0,Y 481.644,Z 245.486,A -85,B 0,C 180,E1 -6869.743,E2 -6869.743} C_VEL
LIN {X 0,Y 481.661,Z 245.486,A -85,B 0,C 180,E1 -6872.675,E2 -6872.675} C_VEL
LIN {X 0,Y 481.611,Z 245.49,A -85,B 0,C 180,E1 -6875.712,E2 -6875.712} C_VEL
LIN {X 0,Y 481.626,Z 245.488,A -85,B 0,C 180,E1 -6878.863,E2 -6878.863} C_VEL
LIN {X 0,Y 481.616,Z 245.49,A -85,B 0,C 180,E1 -6881.909,E2 -6881.909} C_VEL
LIN {X 0,Y 481.646,Z 245.488,A -85,B 0,C 180,E1 -6884.459,E2 -6884.459} C_VEL
LIN {X 0,Y 481.607,Z 245.494,A -85,B 0,C 180,E1 -6886.856,E2 -6886.856} C_VEL
LIN {X 0,Y 481.625,Z 245.485,A -85,B 0,C 180,E1 -6890.055,E2 -6890.055} C_VEL
LIN {X 0,Y 481.599,Z 245.494,A -85,B 0,C 180,E1 -6893.251,E2 -6893.251} C_VEL
LIN {X 0,Y 481.669,Z 245.486,A -85,B 0,C 180,E1 -6896.327,E2 -6896.327} C_VEL
LIN {X 0,Y 481.609,Z 245.495,A -85,B 0,C 180,E1 -6899.426,E2 -6899.426} C_VEL
LIN {X 0,Y 481.668,Z 245.674,A -85,B 0,C 180,E1 -6901.086,E2 -6901.086} C_VEL
LIN {X 0,Y 484.39,Z 258.642,A -85,B 0,C 180,E1 -6903.057,E2 -6903.057} C_VEL
LIN {X 0,Y 484.356,Z 265.395,A -85,B 0,C 180,E1 -6903.988,E2 -6903.988} C_VEL
LIN {X 0,Y 483.622,Z 286.97,A -85,B 0,C 180,E1 -6906.898,E2 -6906.898} C_VEL
LIN {X 0,Y 482.911,Z 308.632,A -85,B 0,C 180,E1 -6909.779,E2 -6909.779} C_VEL
LIN {X 0,Y 482.346,Z 330.228,A -85,B 0,C 180,E1 -6912.621,E2 -6912.621} C_VEL
LIN {X 0,Y 482.21,Z 336.287,A -85,B 0,C 180,E1 -6913.396,E2 -6913.396} C_VEL
LIN {X 0,Y 484.083,Z 352.818,A -85,B 0,C 180,E1 -6913.743,E2 -6913.743} C_VEL
LIN {X 0,Y 484.764,Z 360.278,A -85,B 0,C 180,E1 -6913.88,E2 -6913.88} C_VEL
LIN {X 0,Y 484.129,Z 447.425,A -85,B 0,C 180,E1 -6915.202,E2 -6915.202} C_VEL
LIN {X 0,Y 483.782,Z 460.493,A -85,B 0,C 180,E1 -6915.568,E2 -6915.568} C_VEL
LIN {X 0,Y 483.329,Z 472.589,A -85,B 0,C 180,E1 -6916.064,E2 -6916.064} C_VEL
LIN {X 0,Y 482.813,Z 484.862,A -85,B 0,C 180,E1 -6916.746,E2 -6916.746} C_VEL
LIN {X 0,Y 482.386,Z 496.856,A -85,B 0,C 180,E1 -6917.616,E2 -6917.616} C_VEL
LIN {X 0,Y 481.898,Z 508.139,A -85,B 0,C 180,E1 -6918.645,E2 -6918.645} C_VEL
LIN {X 0,Y 481.547,Z 517.434,A -85,B 0,C 180,E1 -6919.701,E2 -6919.701} C_VEL
LIN {X 0,Y 481.293,Z 526.529,A -85,B 0,C 180,E1 -6920.968,E2 -6920.968} C_VEL
LIN {X 0,Y 481.139,Z 533.871,A -85,B 0,C 180,E1 -6922.235,E2 -6922.235} C_VEL
LIN {X 0,Y 481.023,Z 539.639,A -85,B 0,C 180,E1 -6923.473,E2 -6923.473} C_VEL
LIN {X 0,Y 481.029,Z 543.679,A -85,B 0,C 180,E1 -6924.55,E2 -6924.55} C_VEL
LIN {X 0,Y 481.069,Z 547.391,A -85,B 0,C 180,E1 -6925.811,E2 -6925.811} C_VEL
LIN {X 0,Y 481.09,Z 549.309,A -85,B 0,C 180,E1 -6926.65,E2 -6926.65} C_VEL
LIN {X 0,Y 481.024,Z 550.739,A -85,B 0,C 180,E1 -6927.488,E2 -6927.488} C_VEL
LIN {X 0,Y 481,Z 552.395,A -85,B 0,C 180,E1 -6929.162,E2 -6929.162} C_VEL
LIN {X 0,Y 481.015,Z 552.625,A -85,B 0,C 180,E1 -6930,E2 -6930} C_VEL
LIN {X 0,Y 480.999,Z 552.408,A -85,B 0,C 180,E1 -6930.837,E2 -6930.837} C_VEL
LIN {X 0,Y 481.02,Z 550.782,A -85,B 0,C 180,E1 -6932.512,E2 -6932.512} C_VEL
LIN {X 0,Y 481.088,Z 549.364,A -85,B 0,C 180,E1 -6933.35,E2 -6933.35} C_VEL
LIN {X 0,Y 481.04,Z 546.358,A -85,B 0,C 180,E1 -6934.609,E2 -6934.609} C_VEL
LIN {X 0,Y 481.061,Z 542.297,A -85,B 0,C 180,E1 -6935.869,E2 -6935.869} C_VEL
LIN {X 0,Y 481.092,Z 537.07,A -85,B 0,C 180,E1 -6937.132,E2 -6937.132} C_VEL
LIN {X 0,Y 481.184,Z 530.489,A -85,B 0,C 180,E1 -6938.398,E2 -6938.398} C_VEL
LIN {X 0,Y 481.382,Z 522.302,A -85,B 0,C 180,E1 -6939.665,E2 -6939.665} C_VEL
LIN {X 0,Y 481.687,Z 513.978,A -85,B 0,C 180,E1 -6940.72,E2 -6940.72} C_VEL
LIN {X 0,Y 482.082,Z 503.839,A -85,B 0,C 180,E1 -6941.776,E2 -6941.776} C_VEL
LIN {X 0,Y 482.527,Z 492.383,A -85,B 0,C 180,E1 -6942.726,E2 -6942.726} C_VEL
LIN {X 0,Y 482.904,Z 481.17,A -85,B 0,C 180,E1 -6943.465,E2 -6943.465} C_VEL
LIN {X 0,Y 483.411,Z 468.755,A -85,B 0,C 180,E1 -6944.094,E2 -6944.094} C_VEL
LIN {X 0,Y 483.854,Z 455.607,A -85,B 0,C 180,E1 -6944.564,E2 -6944.564} C_VEL
LIN {X 0,Y 484.154,Z 443.035,A -85,B 0,C 180,E1 -6944.85,E2 -6944.85} C_VEL
LIN {X 0,Y 484.586,Z 357.862,A -85,B 0,C 180,E1 -6946.114,E2 -6946.114} C_VEL
LIN {X 0,Y 482.24,Z 337.107,A -85,B 0,C 180,E1 -6946.51,E2 -6946.51} C_VEL
LIN {X 0,Y 482.257,Z 333.372,A -85,B 0,C 180,E1 -6946.945,E2 -6946.945} C_VEL
LIN {X 0,Y 482.841,Z 311.66,A -85,B 0,C 180,E1 -6949.78,E2 -6949.78} C_VEL
LIN {X 0,Y 483.529,Z 286.363,A -85,B 0,C 180,E1 -6953.105,E2 -6953.105} C_VEL
LIN {X 0,Y 484.23,Z 264.425,A -85,B 0,C 180,E1 -6956.018,E2 -6956.018} C_VEL
LIN {X 0,Y 484.128,Z 257.572,A -85,B 0,C 180,E1 -6956.948,E2 -6956.948} C_VEL
LIN {X 0,Y 481.641,Z 245.663,A -85,B 0,C 180,E1 -6958.695,E2 -6958.695} C_VEL
LIN {X 0,Y 481.617,Z 245.496,A -85,B 0,C 180,E1 -6961.689,E2 -6961.689} C_VEL
LIN {X 0,Y 481.672,Z 245.484,A -85,B 0,C 180,E1 -6964.682,E2 -6964.682} C_VEL
LIN {X 0,Y 481.615,Z 245.489,A -85,B 0,C 180,E1 -6968.001,E2 -6968.001} C_VEL
LIN {X 0,Y 481.605,Z 245.494,A -85,B 0,C 180,E1 -6971.045,E2 -6971.045} C_VEL
LIN {X 0,Y 481.641,Z 245.485,A -85,B 0,C 180,E1 -6974.458,E2 -6974.458} C_VEL
LIN {X 0,Y 481.603,Z 245.493,A -85,B 0,C 180,E1 -6976.855,E2 -6976.855} C_VEL
LIN {X 0,Y 481.646,Z 245.484,A -85,B 0,C 180,E1 -6980.056,E2 -6980.056} C_VEL
LIN {X 0,Y 481.598,Z 245.495,A -85,B 0,C 180,E1 -6983.379,E2 -6983.379} C_VEL
LIN {X 0,Y 481.66,Z 245.483,A -85,B 0,C 180,E1 -6986.326,E2 -6986.326} C_VEL
LIN {X 0,Y 481.615,Z 245.491,A -85,B 0,C 180,E1 -6989.422,E2 -6989.422} C_VEL
LIN {X 0,Y 481.633,Z 245.486,A -85,B 0,C 180,E1 -6992.164,E2 -6992.164} C_VEL
LIN {X 0,Y 481.654,Z 245.491,A -85,B 0,C 180,E1 -6994.966,E2 -6994.966} C_VEL
LIN {X 0,Y 481.632,Z 245.486,A -85,B 0,C 180,E1 -6997.704,E2 -6997.704} C_VEL
LIN {X 0,Y 481.679,Z 245.483,A -85,B 0,C 180,E1 -7000.392,E2 -7000.392} C_VEL
LIN {X 0,Y 481.646,Z 245.489,A -85,B 0,C 180,E1 -7003.032,E2 -7003.032} C_VEL
LIN {X 0,Y 481.654,Z 245.483,A -85,B 0,C 180,E1 -7005.638,E2 -7005.638} C_VEL
LIN {X 0,Y 481.736,Z 245.475,A -85,B 0,C 180,E1 -7008.215,E2 -7008.215} C_VEL
LIN {X 0,Y 481.704,Z 245.477,A -85,B 0,C 180,E1 -7011.611,E2 -7011.611} C_VEL
LIN {X 0,Y 481.75,Z 245.474,A -85,B 0,C 180,E1 -7014.139,E2 -7014.139} C_VEL
LIN {X 0,Y 481.899,Z 245.453,A -85,B 0,C 180,E1 -7017.493,E2 -7017.493} C_VEL
LIN {X 0,Y 481.831,Z 245.465,A -85,B 0,C 180,E1 -7020.836,E2 -7020.836} C_VEL
LIN {X 0,Y 481.89,Z 245.462,A -85,B 0,C 180,E1 -7022.508,E2 -7022.508} C_VEL
LIN {X 0,Y 481.759,Z 245.472,A -85,B 0,C 180,E1 -7025.861,E2 -7025.861} C_VEL
LIN {X 0,Y 481.698,Z 245.486,A -85,B 0,C 180,E1 -7028.39,E2 -7028.39} C_VEL
LIN {X 0,Y 481.72,Z 245.477,A -85,B 0,C 180,E1 -7031.786,E2 -7031.786} C_VEL
LIN {X 0,Y 481.727,Z 245.474,A -85,B 0,C 180,E1 -7035.225,E2 -7035.225} C_VEL
LIN {X 0,Y 481.692,Z 245.48,A -85,B 0,C 180,E1 -7038.723,E2 -7038.723} C_VEL
LIN {X 0,Y 481.632,Z 245.486,A -85,B 0,C 180,E1 -7041.396,E2 -7041.396} C_VEL
LIN {X 0,Y 481.636,Z 245.494,A -85,B 0,C 180,E1 -7044.116,E2 -7044.116} C_VEL
LIN {X 0,Y 481.639,Z 245.485,A -85,B 0,C 180,E1 -7047.117,E2 -7047.117} C_VEL
LIN {X 0,Y 481.654,Z 245.488,A -85,B 0,C 180,E1 -7049.743,E2 -7049.743} C_VEL
LIN {X 0,Y 481.638,Z 245.486,A -85,B 0,C 180,E1 -7052.677,E2 -7052.677} C_VEL
LIN {X 0,Y 481.64,Z 245.486,A -85,B 0,C 180,E1 -7055.203,E2 -7055.203} C_VEL
LIN {X 0,Y 481.617,Z 245.495,A -85,B 0,C 180,E1 -7058.004,E2 -7058.004} C_VEL
LIN {X 0,Y 481.596,Z 245.491,A -85,B 0,C 180,E1 -7061.049,E2 -7061.049} C_VEL
LIN {X 0,Y 481.643,Z 245.485,A -85,B 0,C 180,E1 -7064.46,E2 -7064.46} C_VEL
LIN {X 0,Y 481.607,Z 245.489,A -85,B 0,C 180,E1 -7066.857,E2 -7066.857} C_VEL
LIN {X 0,Y 481.624,Z 245.49,A -85,B 0,C 180,E1 -7070.056,E2 -7070.056} C_VEL
LIN {X 0,Y 481.6,Z 245.493,A -85,B 0,C 180,E1 -7073.252,E2 -7073.252} C_VEL
LIN {X 0,Y 481.668,Z 245.482,A -85,B 0,C 180,E1 -7076.328,E2 -7076.328} C_VEL
LIN {X 0,Y 481.61,Z 245.496,A -85,B 0,C 180,E1 -7079.427,E2 -7079.427} C_VEL
LIN {X 0,Y 481.641,Z 245.486,A -85,B 0,C 180,E1 -7082.165,E2 -7082.165} C_VEL
LIN {X 0,Y 481.665,Z 245.484,A -85,B 0,C 180,E1 -7084.968,E2 -7084.968} C_VEL
LIN {X 0,Y 481.624,Z 245.488,A -85,B 0,C 180,E1 -7087.988,E2 -7087.988} C_VEL
LIN {X 0,Y 480.957,Z 245.572,A -85,B 0,C 180,E1 -7088.686,E2 -7088.686} C_VEL
LIN {X 0,Y 478.123,Z 245.929,A -85,B 0,C 180,E1 -7089.819,E2 -7089.819} C_VEL
LIN {X 0,Y 475.729,Z 246.23,A -85,B 0,C 180,E1 -7090.733,E2 -7090.733} C_VEL
LIN {X 0,Y 474.703,Z 246.356,A -85,B 0,C 180,E1 -7091.439,E2 -7091.439} C_VEL
LIN {X 0,Y 474.62,Z 246.363,A -85,B 0,C 180,E1 -7091.678,E2 -7091.678} C_VEL
LIN {X 0,Y 474.652,Z 246.356,A -85,B 0,C 180,E1 -7094.543,E2 -7094.543} C_VEL
LIN {X 0,Y 474.696,Z 246.352,A -85,B 0,C 180,E1 -7098.038,E2 -7098.038} C_VEL
LIN {X 0,Y 474.686,Z 246.496,A -85,B 0,C 180,E1 -7101.486,E2 -7101.486} C_VEL
LIN {X 0,Y 474.911,Z 247.498,A -85,B 0,C 180,E1 -7101.639,E2 -7101.639} C_VEL
LIN {X 0,Y 478.069,Z 256.367,A -85,B 0,C 180,E1 -7101.896,E2 -7101.896} C_VEL
LIN {X 0,Y 477.595,Z 335.111,A -85,B 0,C 180,E1 -7103.107,E2 -7103.107} C_VEL
LIN {X 0,Y 477.478,Z 348.768,A -85,B 0,C 180,E1 -7103.503,E2 -7103.503} C_VEL
LIN {X 0,Y 477.283,Z 361.032,A -85,B 0,C 180,E1 -7104.031,E2 -7104.031} C_VEL
LIN {X 0,Y 476.973,Z 372.786,A -85,B 0,C 180,E1 -7104.717,E2 -7104.717} C_VEL
LIN {X 0,Y 476.54,Z 384.042,A -85,B 0,C 180,E1 -7105.56,E2 -7105.56} C_VEL
LIN {X 0,Y 476.129,Z 394.183,A -85,B 0,C 180,E1 -7106.51,E2 -7106.51} C_VEL
LIN {X 0,Y 475.757,Z 402.484,A -85,B 0,C 180,E1 -7107.46,E2 -7107.46} C_VEL
LIN {X 0,Y 475.427,Z 410.142,A -85,B 0,C 180,E1 -7108.518,E2 -7108.518} C_VEL
LIN {X 0,Y 475.004,Z 417.653,A -85,B 0,C 180,E1 -7109.788,E2 -7109.788} C_VEL
LIN {X 0,Y 474.662,Z 424.568,A -85,B 0,C 180,E1 -7111.273,E2 -7111.273} C_VEL
LIN {X 0,Y 474.51,Z 429.165,A -85,B 0,C 180,E1 -7112.547,E2 -7112.547} C_VEL
LIN {X 0,Y 474.378,Z 431.653,A -85,B 0,C 180,E1 -7113.398,E2 -7113.398} C_VEL
LIN {X 0,Y 474.323,Z 433.647,A -85,B 0,C 180,E1 -7114.249,E2 -7114.249} C_VEL
LIN {X 0,Y 474.324,Z 435.231,A -85,B 0,C 180,E1 -7115.101,E2 -7115.101} C_VEL
LIN {X 0,Y 474.29,Z 436.432,A -85,B 0,C 180,E1 -7115.954,E2 -7115.954} C_VEL
LIN {X 0,Y 474.268,Z 437.237,A -85,B 0,C 180,E1 -7116.852,E2 -7116.852} C_VEL
LIN {X 0,Y 474.203,Z 437.603,A -85,B 0,C 180,E1 -7118.523,E2 -7118.523} C_VEL
LIN {X 0,Y 474.219,Z 437.229,A -85,B 0,C 180,E1 -7119.382,E2 -7119.382} C_VEL
LIN {X 0,Y 474.218,Z 436.431,A -85,B 0,C 180,E1 -7120.244,E2 -7120.244} C_VEL
LIN {X 0,Y 474.335,Z 435.21,A -85,B 0,C 180,E1 -7121.106,E2 -7121.106} C_VEL
LIN {X 0,Y 474.412,Z 433.307,A -85,B 0,C 180,E1 -7122.111,E2 -7122.111} C_VEL
LIN {X 0,Y 474.6,Z 428.98,A -85,B 0,C 180,E1 -7123.706,E2 -7123.706} C_VEL
LIN {X 0,Y 474.843,Z 424.199,A -85,B 0,C 180,E1 -7125.011,E2 -7125.011} C_VEL
LIN {X 0,Y 475.145,Z 418.112,A -85,B 0,C 180,E1 -7126.322,E2 -7126.322} C_VEL
LIN {X 0,Y 475.543,Z 410.471,A -85,B 0,C 180,E1 -7127.636,E2 -7127.636} C_VEL
LIN {X 0,Y 475.948,Z 402.56,A -85,B 0,C 180,E1 -7128.733,E2 -7128.733} C_VEL
LIN {X 0,Y 476.385,Z 392.824,A -85,B 0,C 180,E1 -7129.835,E2 -7129.835} C_VEL
LIN {X 0,Y 476.808,Z 381.908,A -85,B 0,C 180,E1 -7130.83,E2 -7130.83} C_VEL
LIN {X 0,Y 477.275,Z 371.138,A -85,B 0,C 180,E1 -7131.6,E2 -7131.6} C_VEL
LIN {X 0,Y 477.59,Z 358.476,A -85,B 0,C 180,E1 -7132.301,E2 -7132.301} C_VEL
LIN {X 0,Y 477.768,Z 346.137,A -85,B 0,C 180,E1 -7132.8,E2 -7132.8} C_VEL
LIN {X 0,Y 477.928,Z 333.231,A -85,B 0,C 180,E1 -7133.135,E2 -7133.135} C_VEL
LIN {X 0,Y 478.385,Z 256.699,A -85,B 0,C 180,E1 -7134.317,E2 -7134.317} C_VEL
LIN {X 0,Y 474.814,Z 247.373,A -85,B 0,C 180,E1 -7134.634,E2 -7134.634} C_VEL
LIN {X 0,Y 474.655,Z 246.484,A -85,B 0,C 180,E1 -7134.785,E2 -7134.785} C_VEL
LIN {X 0,Y 474.61,Z 246.364,A -85,B 0,C 180,E1 -7138.284,E2 -7138.284} C_VEL
LIN {X 0,Y 474.599,Z 246.352,A -85,B 0,C 180,E1 -7141.217,E2 -7141.217} C_VEL
LIN {X 0,Y 474.62,Z 246.365,A -85,B 0,C 180,E1 -7144.242,E2 -7144.242} C_VEL
LIN {X 0,Y 474.575,Z 246.355,A -85,B 0,C 180,E1 -7147.385,E2 -7147.385} C_VEL
LIN {X 0,Y 474.6,Z 246.365,A -85,B 0,C 180,E1 -7149.643,E2 -7149.643} C_VEL
LIN {X 0,Y 474.573,Z 246.371,A -85,B 0,C 180,E1 -7152.938,E2 -7152.938} C_VEL
LIN {X 0,Y 474.599,Z 246.364,A -85,B 0,C 180,E1 -7155.893,E2 -7155.893} C_VEL
LIN {X 0,Y 474.588,Z 246.365,A -85,B 0,C 180,E1 -7159.339,E2 -7159.339} C_VEL
LIN {X 0,Y 474.587,Z 246.36,A -85,B 0,C 180,E1 -7161.706,E2 -7161.706} C_VEL
LIN {X 0,Y 474.612,Z 246.366,A -85,B 0,C 180,E1 -7164.724,E2 -7164.724} C_VEL
LIN {X 0,Y 474.631,Z 246.36,A -85,B 0,C 180,E1 -7167.787,E2 -7167.787} C_VEL
LIN {X 0,Y 474.597,Z 246.359,A -85,B 0,C 180,E1 -7170.889,E2 -7170.889} C_VEL
LIN {X 0,Y 474.587,Z 246.367,A -85,B 0,C 180,E1 -7173.624,E2 -7173.624} C_VEL
LIN {X 0,Y 474.629,Z 246.349,A -85,B 0,C 180,E1 -7176.641,E2 -7176.641} C_VEL
LIN {X 0,Y 474.646,Z 246.352,A -85,B 0,C 180,E1 -7180.089,E2 -7180.089} C_VEL
LIN {X 0,Y 474.626,Z 246.36,A -85,B 0,C 180,E1 -7182.773,E2 -7182.773} C_VEL
LIN {X 0,Y 474.633,Z 246.357,A -85,B 0,C 180,E1 -7185.42,E2 -7185.42} C_VEL
LIN {X 0,Y 474.697,Z 246.356,A -85,B 0,C 180,E1 -7188.037,E2 -7188.037} C_VEL
LIN {X 0,Y 474.688,Z 246.349,A -85,B 0,C 180,E1 -7191.486,E2 -7191.486} C_VEL
LIN {X 0,Y 474.73,Z 246.349,A -85,B 0,C 180,E1 -7194.052,E2 -7194.052} C_VEL
LIN {X 0,Y 474.863,Z 246.33,A -85,B 0,C 180,E1 -7197.455,E2 -7197.455} C_VEL
LIN {X 0,Y 474.87,Z 246.331,A -85,B 0,C 180,E1 -7200,E2 -7200} C_VEL
LIN {X 0,Y 474.872,Z 246.325,A -85,B 0,C 180,E1 -7202.545,E2 -7202.545} C_VEL
LIN {X 0,Y 474.72,Z 246.348,A -85,B 0,C 180,E1 -7205.948,E2 -7205.948} C_VEL
LIN {X 0,Y 474.698,Z 246.347,A -85,B 0,C 180,E1 -7208.514,E2 -7208.514} C_VEL
LIN {X 0,Y 474.696,Z 246.349,A -85,B 0,C 180,E1 -7211.963,E2 -7211.963} C_VEL
LIN {X 0,Y 474.671,Z 246.357,A -85,B 0,C 180,E1 -7215.767,E2 -7215.767} C_VEL
LIN {X 0,Y 474.652,Z 246.358,A -85,B 0,C 180,E1 -7219.011,E2 -7219.011} C_VEL
LIN {X 0,Y 474.58,Z 246.365,A -85,B 0,C 180,E1 -7221.729,E2 -7221.729} C_VEL
LIN {X 0,Y 474.618,Z 246.362,A -85,B 0,C 180,E1 -7224.495,E2 -7224.495} C_VEL
LIN {X 0,Y 474.59,Z 246.358,A -85,B 0,C 180,E1 -7227.327,E2 -7227.327} C_VEL
LIN {X 0,Y 474.574,Z 246.366,A -85,B 0,C 180,E1 -7230.232,E2 -7230.232} C_VEL
LIN {X 0,Y 474.615,Z 246.357,A -85,B 0,C 180,E1 -7233.222,E2 -7233.222} C_VEL
LIN {X 0,Y 474.566,Z 246.369,A -85,B 0,C 180,E1 -7236.326,E2 -7236.326} C_VEL
LIN {X 0,Y 474.595,Z 246.363,A -85,B 0,C 180,E1 -7239.644,E2 -7239.644} C_VEL
LIN {X 0,Y 474.57,Z 246.369,A -85,B 0,C 180,E1 -7242.23,E2 -7242.23} C_VEL
LIN {X 0,Y 474.608,Z 246.364,A -85,B 0,C 180,E1 -7245.299,E2 -7245.299} C_VEL
LIN {X 0,Y 474.586,Z 246.368,A -85,B 0,C 180,E1 -7248.212,E2 -7248.212} C_VEL
LIN {X 0,Y 474.578,Z 246.363,A -85,B 0,C 180,E1 -7251.54,E2 -7251.54} C_VEL
LIN {X 0,Y 474.607,Z 246.359,A -85,B 0,C 180,E1 -7254.725,E2 -7254.725} C_VEL
LIN {X 0,Y 474.615,Z 246.359,A -85,B 0,C 180,E1 -7257.787,E2 -7257.787} C_VEL
LIN {X 0,Y 474.628,Z 246.613,A -85,B 0,C 180,E1 -7260.854,E2 -7260.854} C_VEL
LIN {X 0,Y 477.412,Z 259.499,A -85,B 0,C 180,E1 -7262.848,E2 -7262.848} C_VEL
LIN {X 0,Y 477.564,Z 264.554,A -85,B 0,C 180,E1 -7263.566,E2 -7263.566} C_VEL
LIN {X 0,Y 476.713,Z 286.271,A -85,B 0,C 180,E1 -7266.544,E2 -7266.544} C_VEL
LIN {X 0,Y 475.992,Z 307.915,A -85,B 0,C 180,E1 -7269.472,E2 -7269.472} C_VEL
LIN {X 0,Y 475.371,Z 329.489,A -85,B 0,C 180,E1 -7272.358,E2 -7272.358} C_VEL
LIN {X 0,Y 475.236,Z 335.612,A -85,B 0,C 180,E1 -7273.141,E2 -7273.141} C_VEL
LIN {X 0,Y 477.971,Z 360.016,A -85,B 0,C 180,E1 -7273.637,E2 -7273.637} C_VEL
LIN {X 0,Y 477.304,Z 446.089,A -85,B 0,C 180,E1 -7274.959,E2 -7274.959} C_VEL
LIN {X 0,Y 476.927,Z 459.3,A -85,B 0,C 180,E1 -7275.329,E2 -7275.329} C_VEL
LIN {X 0,Y 476.434,Z 470.901,A -85,B 0,C 180,E1 -7275.804,E2 -7275.804} C_VEL
LIN {X 0,Y 475.961,Z 482.542,A -85,B 0,C 180,E1 -7276.443,E2 -7276.443} C_VEL
LIN {X 0,Y 475.481,Z 493.205,A -85,B 0,C 180,E1 -7277.19,E2 -7277.19} C_VEL
LIN {X 0,Y 475.033,Z 504.169,A -85,B 0,C 180,E1 -7278.154,E2 -7278.154} C_VEL
LIN {X 0,Y 474.66,Z 513.147,A -85,B 0,C 180,E1 -7279.118,E2 -7279.118} C_VEL
LIN {X 0,Y 474.283,Z 522.935,A -85,B 0,C 180,E1 -7280.404,E2 -7280.404} C_VEL
LIN {X 0,Y 474.098,Z 530.764,A -85,B 0,C 180,E1 -7281.69,E2 -7281.69} C_VEL
LIN {X 0,Y 473.977,Z 538.007,A -85,B 0,C 180,E1 -7283.187,E2 -7283.187} C_VEL
LIN {X 0,Y 473.966,Z 542.842,A -85,B 0,C 180,E1 -7284.469,E2 -7284.469} C_VEL
LIN {X 0,Y 474.009,Z 546.549,A -85,B 0,C 180,E1 -7285.748,E2 -7285.748} C_VEL
LIN {X 0,Y 474.039,Z 548.465,A -85,B 0,C 180,E1 -7286.6,E2 -7286.6} C_VEL
LIN {X 0,Y 473.967,Z 549.892,A -85,B 0,C 180,E1 -7287.45,E2 -7287.45} C_VEL
LIN {X 0,Y 473.948,Z 551.548,A -85,B 0,C 180,E1 -7289.15,E2 -7289.15} C_VEL
LIN {X 0,Y 473.966,Z 551.776,A -85,B 0,C 180,E1 -7290,E2 -7290} C_VEL
LIN {X 0,Y 473.948,Z 551.557,A -85,B 0,C 180,E1 -7290.849,E2 -7290.849} C_VEL
LIN {X 0,Y 473.965,Z 549.927,A -85,B 0,C 180,E1 -7292.549,E2 -7292.549} C_VEL
LIN {X 0,Y 474.037,Z 548.507,A -85,B 0,C 180,E1 -7293.399,E2 -7293.399} C_VEL
LIN {X 0,Y 473.961,Z 545.493,A -85,B 0,C 180,E1 -7294.678,E2 -7294.678} C_VEL
LIN {X 0,Y 473.952,Z 540.329,A -85,B 0,C 180,E1 -7296.244,E2 -7296.244} C_VEL
LIN {X 0,Y 474.03,Z 534.122,A -85,B 0,C 180,E1 -7297.668,E2 -7297.668} C_VEL
LIN {X 0,Y 474.187,Z 527.064,A -85,B 0,C 180,E1 -7298.952,E2 -7298.952} C_VEL
LIN {X 0,Y 474.431,Z 518.232,A -85,B 0,C 180,E1 -7300.239,E2 -7300.239} C_VEL
LIN {X 0,Y 474.842,Z 508.21,A -85,B 0,C 180,E1 -7301.417,E2 -7301.417} C_VEL
LIN {X 0,Y 475.32,Z 498.307,A -85,B 0,C 180,E1 -7302.361,E2 -7302.361} C_VEL
LIN {X 0,Y 475.713,Z 486.858,A -85,B 0,C 180,E1 -7303.237,E2 -7303.237} C_VEL
LIN {X 0,Y 476.242,Z 474.297,A -85,B 0,C 180,E1 -7303.983,E2 -7303.983} C_VEL
LIN {X 0,Y 476.725,Z 461.595,A -85,B 0,C 180,E1 -7304.541,E2 -7304.541} C_VEL
LIN {X 0,Y 477.13,Z 448.126,A -85,B 0,C 180,E1 -7304.937,E2 -7304.937} C_VEL
LIN {X 0,Y 477.312,Z 423.543,A -85,B 0,C 180,E1 -7305.341,E2 -7305.341} C_VEL
LIN {X 0,Y 477.711,Z 358.549,A -85,B 0,C 180,E1 -7306.317,E2 -7306.317} C_VEL
LIN {X 0,Y 475.19,Z 335.858,A -85,B 0,C 180,E1 -7306.762,E2 -7306.762} C_VEL
LIN {X 0,Y 475.825,Z 312.323,A -85,B 0,C 180,E1 -7309.859,E2 -7309.859} C_VEL
LIN {X 0,Y 476.495,Z 288.705,A -85,B 0,C 180,E1 -7313.007,E2 -7313.007} C_VEL
LIN {X 0,Y 477.174,Z 268.594,A -85,B 0,C 180,E1 -7315.711,E2 -7315.711} C_VEL
LIN {X 0,Y 477.297,Z 259.705,A -85,B 0,C 180,E1 -7316.921,E2 -7316.921} C_VEL
LIN {X 0,Y 474.587,Z 246.5,A -85,B 0,C 180,E1 -7318.892,E2 -7318.892} C_VEL
LIN {X 0,Y 474.612,Z 246.364,A -85,B 0,C 180,E1 -7322.213,E2 -7322.213} C_VEL
LIN {X 0,Y 474.604,Z 246.369,A -85,B 0,C 180,E1 -7325.275,E2 -7325.275} C_VEL
LIN {X 0,Y 474.575,Z 246.365,A -85,B 0,C 180,E1 -7328.459,E2 -7328.459} C_VEL
LIN {X 0,Y 474.582,Z 246.367,A -85,B 0,C 180,E1 -7331.788,E2 -7331.788} C_VEL
LIN {X 0,Y 474.604,Z 246.369,A -85,B 0,C 180,E1 -7335.297,E2 -7335.297} C_VEL
LIN {X 0,Y 474.582,Z 246.364,A -85,B 0,C 180,E1 -7338.21,E2 -7338.21} C_VEL
LIN {X 0,Y 474.588,Z 246.367,A -85,B 0,C 180,E1 -7341.54,E2 -7341.54} C_VEL
LIN {X 0,Y 474.599,Z 246.366,A -85,B 0,C 180,E1 -7344.723,E2 -7344.723} C_VEL
LIN {X 0,Y 474.598,Z 246.363,A -85,B 0,C 180,E1 -7347.785,E2 -7347.785} C_VEL
LIN {X 0,Y 474.581,Z 246.372,A -85,B 0,C 180,E1 -7350.891,E2 -7350.891} C_VEL
LIN {X 0,Y 474.559,Z 246.368,A -85,B 0,C 180,E1 -7353.622,E2 -7353.622} C_VEL
